LIN {X 0,Y 319.551,Z 618.351,A -85,B 0,C 180,E1 -16134.442,E2 -16134.442} C_VEL
LIN {X 0,Y 320.953,Z 553.396,A -85,B 0,C 180,E1 -16135.793,E2 -16135.793} C_VEL
LIN {X 0,Y 315.824,Z 527.025,A -85,B 0,C 180,E1 -16136.903,E2 -16136.903} C_VEL
LIN {X 0,Y 313.35,Z 517.185,A -85,B 0,C 180,E1 -16137.39,E2 -16137.39} C_VEL
LIN {X 0,Y 311.493,Z 507.907,A -85,B 0,C 180,E1 -16140.123,E2 -16140.123} C_VEL
LIN {X 0,Y 309.031,Z 497.224,A -85,B 0,C 180,E1 -16143.471,E2 -16143.471} C_VEL
LIN {X 0,Y 306.128,Z 486.248,A -85,B 0,C 180,E1 -16147.182,E2 -16147.182} C_VEL
LIN {X 0,Y 305.497,Z 484.053,A -85,B 0,C 180,E1 -16147.997,E2 -16147.997} C_VEL
LIN {X 0,Y 304.829,Z 484.139,A -85,B 0,C 180,E1 -16149.096,E2 -16149.096} C_VEL
LIN {X 0,Y 301.96,Z 484.493,A -85,B 0,C 180,E1 -16150.885,E2 -16150.885} C_VEL
LIN {X 0,Y 299.514,Z 484.803,A -85,B 0,C 180,E1 -16152.335,E2 -16152.335} C_VEL
LIN {X 0,Y 298.446,Z 484.931,A -85,B 0,C 180,E1 -16153.459,E2 -16153.459} C_VEL
LIN {X 0,Y 298.35,Z 484.939,A -85,B 0,C 180,E1 -16153.841,E2 -16153.841} C_VEL
LIN {X 0,Y 298.409,Z 484.934,A -85,B 0,C 180,E1 -16156.921,E2 -16156.921} C_VEL
LIN {X 0,Y 298.405,Z 484.931,A -85,B 0,C 180,E1 -16161.008,E2 -16161.008} C_VEL
LIN {X 0,Y 298.425,Z 484.937,A -85,B 0,C 180,E1 -16163.931,E2 -16163.931} C_VEL
LIN {X 0,Y 298.49,Z 485.123,A -85,B 0,C 180,E1 -16166.405,E2 -16166.405} C_VEL
LIN {X 0,Y 302.37,Z 501.908,A -85,B 0,C 180,E1 -16170.085,E2 -16170.085} C_VEL
LIN {X 0,Y 304.66,Z 513.404,A -85,B 0,C 180,E1 -16172.524,E2 -16172.524} C_VEL
LIN {X 0,Y 303.462,Z 529.943,A -85,B 0,C 180,E1 -16175.727,E2 -16175.727} C_VEL
LIN {X 0,Y 303.246,Z 533.339,A -85,B 0,C 180,E1 -16176.367,E2 -16176.367} C_VEL
LIN {X 0,Y 306.285,Z 559.768,A -85,B 0,C 180,E1 -16177.442,E2 -16177.442} C_VEL
LIN {X 0,Y 303.271,Z 645.533,A -85,B 0,C 180,E1 -16180.365,E2 -16180.365} C_VEL
LIN {X 0,Y 302.635,Z 658.135,A -85,B 0,C 180,E1 -16181.027,E2 -16181.027} C_VEL
LIN {X 0,Y 301.907,Z 671.811,A -85,B 0,C 180,E1 -16182.034,E2 -16182.034} C_VEL
LIN {X 0,Y 300.975,Z 684.908,A -85,B 0,C 180,E1 -16183.311,E2 -16183.311} C_VEL
LIN {X 0,Y 300.064,Z 696.338,A -85,B 0,C 180,E1 -16184.722,E2 -16184.722} C_VEL
LIN {X 0,Y 299.145,Z 707.277,A -85,B 0,C 180,E1 -16186.412,E2 -16186.412} C_VEL
LIN {X 0,Y 298.382,Z 716.255,A -85,B 0,C 180,E1 -16188.106,E2 -16188.106} C_VEL
LIN {X 0,Y 297.71,Z 725.006,A -85,B 0,C 180,E1 -16190.145,E2 -16190.145} C_VEL
LIN {X 0,Y 297.211,Z 732.04,A -85,B 0,C 180,E1 -16192.185,E2 -16192.185} C_VEL
LIN {X 0,Y 296.865,Z 737.87,A -85,B 0,C 180,E1 -16194.322,E2 -16194.322} C_VEL
LIN {X 0,Y 296.754,Z 742.533,A -85,B 0,C 180,E1 -16196.605,E2 -16196.605} C_VEL
LIN {X 0,Y 296.627,Z 745.53,A -85,B 0,C 180,E1 -16198.642,E2 -16198.642} C_VEL
LIN {X 0,Y 296.633,Z 746.97,A -85,B 0,C 180,E1 -16200,E2 -16200} C_VEL
LIN {X 0,Y 296.755,Z 747.956,A -85,B 0,C 180,E1 -16201.357,E2 -16201.357} C_VEL
LIN {X 0,Y 296.931,Z 748.483,A -85,B 0,C 180,E1 -16202.713,E2 -16202.713} C_VEL
LIN {X 0,Y 297.089,Z 748.604,A -85,B 0,C 180,E1 -16204.069,E2 -16204.069} C_VEL
LIN {X 0,Y 297.301,Z 748.296,A -85,B 0,C 180,E1 -16205.426,E2 -16205.426} C_VEL
LIN {X 0,Y 297.711,Z 747.521,A -85,B 0,C 180,E1 -16206.778,E2 -16206.778} C_VEL
LIN {X 0,Y 298.406,Z 746.025,A -85,B 0,C 180,E1 -16208.43,E2 -16208.43} C_VEL
LIN {X 0,Y 299.55,Z 742.622,A -85,B 0,C 180,E1 -16210.818,E2 -16210.818} C_VEL
LIN {X 0,Y 300.846,Z 738.565,A -85,B 0,C 180,E1 -16212.822,E2 -16212.822} C_VEL
LIN {X 0,Y 302.734,Z 732.402,A -85,B 0,C 180,E1 -16215.139,E2 -16215.139} C_VEL
LIN {X 0,Y 304.769,Z 725.583,A -85,B 0,C 180,E1 -16217.098,E2 -16217.098} C_VEL
LIN {X 0,Y 306.644,Z 718.669,A -85,B 0,C 180,E1 -16218.715,E2 -16218.715} C_VEL
LIN {X 0,Y 309.275,Z 708.641,A -85,B 0,C 180,E1 -16220.623,E2 -16220.623} C_VEL
LIN {X 0,Y 311.91,Z 697.136,A -85,B 0,C 180,E1 -16222.343,E2 -16222.343} C_VEL
LIN {X 0,Y 314.257,Z 685.303,A -85,B 0,C 180,E1 -16223.738,E2 -16223.738} C_VEL
LIN {X 0,Y 316.279,Z 674.01,A -85,B 0,C 180,E1 -16224.798,E2 -16224.798} C_VEL
LIN {X 0,Y 318.093,Z 661.718,A -85,B 0,C 180,E1 -16225.696,E2 -16225.696} C_VEL
LIN {X 0,Y 319.7,Z 647.864,A -85,B 0,C 180,E1 -16226.433,E2 -16226.433} C_VEL
LIN {X 0,Y 327.907,Z 571.032,A -85,B 0,C 180,E1 -16229.456,E2 -16229.456} C_VEL
LIN {X 0,Y 327.938,Z 568.4,A -85,B 0,C 180,E1 -16229.628,E2 -16229.628} C_VEL
LIN {X 0,Y 326.362,Z 556.568,A -85,B 0,C 180,E1 -16230.828,E2 -16230.828} C_VEL
LIN {X 0,Y 324.446,Z 544.971,A -85,B 0,C 180,E1 -16232.247,E2 -16232.247} C_VEL
LIN {X 0,Y 322.625,Z 540.593,A -85,B 0,C 180,E1 -16233.189,E2 -16233.189} C_VEL
LIN {X 0,Y 322.019,Z 534.22,A -85,B 0,C 180,E1 -16235.642,E2 -16235.642} C_VEL
LIN {X 0,Y 321.293,Z 529.338,A -85,B 0,C 180,E1 -16238.049,E2 -16238.049} C_VEL
LIN {X 0,Y 320.801,Z 526.352,A -85,B 0,C 180,E1 -16239.934,E2 -16239.934} C_VEL
LIN {X 0,Y 320.418,Z 524.32,A -85,B 0,C 180,E1 -16241.774,E2 -16241.774} C_VEL
LIN {X 0,Y 320.289,Z 522.915,A -85,B 0,C 180,E1 -16243.604,E2 -16243.604} C_VEL
LIN {X 0,Y 320.596,Z 522.275,A -85,B 0,C 180,E1 -16246.337,E2 -16246.337} C_VEL
LIN {X 0,Y 321.718,Z 523.09,A -85,B 0,C 180,E1 -16249.052,E2 -16249.052} C_VEL
LIN {X 0,Y 323.484,Z 525.204,A -85,B 0,C 180,E1 -16251.456,E2 -16251.456} C_VEL
LIN {X 0,Y 324.046,Z 526.038,A -85,B 0,C 180,E1 -16252.067,E2 -16252.067} C_VEL
LIN {X 0,Y 324.345,Z 528.935,A -85,B 0,C 180,E1 -16253.107,E2 -16253.107} C_VEL
LIN {X 0,Y 325.342,Z 539.139,A -85,B 0,C 180,E1 -16255.829,E2 -16255.829} C_VEL
LIN {X 0,Y 325.845,Z 542.951,A -85,B 0,C 180,E1 -16256.666,E2 -16256.666} C_VEL
LIN {X 0,Y 325.078,Z 550.225,A -85,B 0,C 180,E1 -16257.605,E2 -16257.605} C_VEL
LIN {X 0,Y 325.069,Z 563.307,A -85,B 0,C 180,E1 -16258.604,E2 -16258.604} C_VEL
LIN {X 0,Y 314.684,Z 654.608,A -85,B 0,C 180,E1 -16262.345,E2 -16262.345} C_VEL
LIN {X 0,Y 312.854,Z 674.382,A -85,B 0,C 180,E1 -16263.256,E2 -16263.256} C_VEL
LIN {X 0,Y 311.102,Z 688.949,A -85,B 0,C 180,E1 -16264.221,E2 -16264.221} C_VEL
LIN {X 0,Y 309.164,Z 702.373,A -85,B 0,C 180,E1 -16265.407,E2 -16265.407} C_VEL
LIN {X 0,Y 307.546,Z 712.736,A -85,B 0,C 180,E1 -16266.562,E2 -16266.562} C_VEL
LIN {X 0,Y 305.364,Z 724.902,A -85,B 0,C 180,E1 -16268.214,E2 -16268.214} C_VEL
LIN {X 0,Y 303.591,Z 733.816,A -85,B 0,C 180,E1 -16269.68,E2 -16269.68} C_VEL
LIN {X 0,Y 301.64,Z 743.646,A -85,B 0,C 180,E1 -16271.665,E2 -16271.665} C_VEL
LIN {X 0,Y 300.077,Z 751.779,A -85,B 0,C 180,E1 -16273.676,E2 -16273.676} C_VEL
LIN {X 0,Y 298.889,Z 758.364,A -85,B 0,C 180,E1 -16275.705,E2 -16275.705} C_VEL
LIN {X 0,Y 297.841,Z 763.736,A -85,B 0,C 180,E1 -16277.737,E2 -16277.737} C_VEL
LIN {X 0,Y 297.203,Z 767.938,A -85,B 0,C 180,E1 -16279.783,E2 -16279.783} C_VEL
LIN {X 0,Y 296.807,Z 771.086,A -85,B 0,C 180,E1 -16281.831,E2 -16281.831} C_VEL
LIN {X 0,Y 296.594,Z 773.62,A -85,B 0,C 180,E1 -16284.396,E2 -16284.396} C_VEL
LIN {X 0,Y 296.64,Z 774.399,A -85,B 0,C 180,E1 -16285.922,E2 -16285.922} C_VEL
LIN {X 0,Y 296.811,Z 774.874,A -85,B 0,C 180,E1 -16289.998,E2 -16289.998} C_VEL
LIN {X 0,Y 296.673,Z 774.112,A -85,B 0,C 180,E1 -16292.714,E2 -16292.714} C_VEL
LIN {X 0,Y 296.687,Z 771.88,A -85,B 0,C 180,E1 -16295.435,E2 -16295.435} C_VEL
LIN {X 0,Y 296.71,Z 769.242,A -85,B 0,C 180,E1 -16297.484,E2 -16297.484} C_VEL
LIN {X 0,Y 297.057,Z 764.251,A -85,B 0,C 180,E1 -16300.219,E2 -16300.219} C_VEL
LIN {X 0,Y 297.678,Z 759.411,A -85,B 0,C 180,E1 -16302.266,E2 -16302.266} C_VEL
LIN {X 0,Y 298.579,Z 752.32,A -85,B 0,C 180,E1 -16304.655,E2 -16304.655} C_VEL
LIN {X 0,Y 299.825,Z 744.889,A -85,B 0,C 180,E1 -16306.685,E2 -16306.685} C_VEL
LIN {X 0,Y 301.331,Z 735.904,A -85,B 0,C 180,E1 -16308.703,E2 -16308.703} C_VEL
LIN {X 0,Y 302.842,Z 726.968,A -85,B 0,C 180,E1 -16310.369,E2 -16310.369} C_VEL
LIN {X 0,Y 304.77,Z 716.28,A -85,B 0,C 180,E1 -16312.005,E2 -16312.005} C_VEL
LIN {X 0,Y 306.67,Z 703.494,A -85,B 0,C 180,E1 -16313.597,E2 -16313.597} C_VEL
LIN {X 0,Y 308.373,Z 691.684,A -85,B 0,C 180,E1 -16314.755,E2 -16314.755} C_VEL
LIN {X 0,Y 310.052,Z 678.252,A -85,B 0,C 180,E1 -16315.778,E2 -16315.778} C_VEL
LIN {X 0,Y 311.401,Z 664.119,A -85,B 0,C 180,E1 -16316.559,E2 -16316.559} C_VEL
LIN {X 0,Y 312.339,Z 650.423,A -85,B 0,C 180,E1 -16317.059,E2 -16317.059} C_VEL
LIN {X 0,Y 315.103,Z 559.841,A -85,B 0,C 180,E1 -16319.246,E2 -16319.246} C_VEL
LIN {X 0,Y 310.597,Z 527.887,A -85,B 0,C 180,E1 -16320.542,E2 -16320.542} C_VEL
LIN {X 0,Y 308.137,Z 521.44,A -85,B 0,C 180,E1 -16320.991,E2 -16320.991} C_VEL
LIN {X 0,Y 305.142,Z 508.508,A -85,B 0,C 180,E1 -16324.478,E2 -16324.478} C_VEL
LIN {X 0,Y 302.125,Z 497.283,A -85,B 0,C 180,E1 -16327.73,E2 -16327.73} C_VEL
LIN {X 0,Y 299.234,Z 487.6,A -85,B 0,C 180,E1 -16330.761,E2 -16330.761} C_VEL
LIN {X 0,Y 298.441,Z 484.935,A -85,B 0,C 180,E1 -16331.699,E2 -16331.699} C_VEL
LIN {X 0,Y 298.482,Z 484.929,A -85,B 0,C 180,E1 -16335.059,E2 -16335.059} C_VEL
LIN {X 0,Y 298.448,Z 484.932,A -85,B 0,C 180,E1 -16338.896,E2 -16338.896} C_VEL
LIN {X 0,Y 298.462,Z 484.907,A -85,B 0,C 180,E1 -16343.185,E2 -16343.185} C_VEL
LIN {X 0,Y 298.388,Z 484.938,A -85,B 0,C 180,E1 -16347.199,E2 -16347.199} C_VEL
LIN {X 0,Y 298.423,Z 484.938,A -85,B 0,C 180,E1 -16350.613,E2 -16350.613} C_VEL
LIN {X 0,Y 298.482,Z 484.929,A -85,B 0,C 180,E1 -16353.47,E2 -16353.47} C_VEL
LIN {X 0,Y 298.42,Z 484.907,A -85,B 0,C 180,E1 -16356.699,E2 -16356.699} C_VEL
LIN {X 0,Y 298.514,Z 484.918,A -85,B 0,C 180,E1 -16360.755,E2 -16360.755} C_VEL
LIN {X 0,Y 298.582,Z 484.911,A -85,B 0,C 180,E1 -16364.994,E2 -16364.994} C_VEL
LIN {X 0,Y 298.585,Z 484.908,A -85,B 0,C 180,E1 -16369.146,E2 -16369.146} C_VEL
LIN {X 0,Y 298.748,Z 484.896,A -85,B 0,C 180,E1 -16371.886,E2 -16371.886} C_VEL
LIN {X 0,Y 298.652,Z 484.9,A -85,B 0,C 180,E1 -16374.599,E2 -16374.599} C_VEL
LIN {X 0,Y 298.915,Z 484.865,A -85,B 0,C 180,E1 -16378.653,E2 -16378.653} C_VEL
LIN {X 0,Y 298.915,Z 484.875,A -85,B 0,C 180,E1 -16381.347,E2 -16381.347} C_VEL
LIN {X 0,Y 298.787,Z 484.889,A -85,B 0,C 180,E1 -16386.754,E2 -16386.754} C_VEL
LIN {X 0,Y 298.67,Z 484.901,A -85,B 0,C 180,E1 -16389.481,E2 -16389.481} C_VEL
LIN {X 0,Y 298.543,Z 484.911,A -85,B 0,C 180,E1 -16393.616,E2 -16393.616} C_VEL
LIN {X 0,Y 298.539,Z 484.921,A -85,B 0,C 180,E1 -16396.409,E2 -16396.409} C_VEL
LIN {X 0,Y 298.502,Z 484.926,A -85,B 0,C 180,E1 -16399.656,E2 -16399.656} C_VEL
LIN {X 0,Y 298.448,Z 484.932,A -85,B 0,C 180,E1 -16403.599,E2 -16403.599} C_VEL
LIN {X 0,Y 298.481,Z 484.922,A -85,B 0,C 180,E1 -16406.576,E2 -16406.576} C_VEL
LIN {X 0,Y 298.417,Z 484.932,A -85,B 0,C 180,E1 -16409.642,E2 -16409.642} C_VEL
LIN {X 0,Y 298.39,Z 484.938,A -85,B 0,C 180,E1 -16412.801,E2 -16412.801} C_VEL
LIN {X 0,Y 298.459,Z 484.927,A -85,B 0,C 180,E1 -16416.814,E2 -16416.814} C_VEL
LIN {X 0,Y 298.412,Z 484.939,A -85,B 0,C 180,E1 -16421.096,E2 -16421.096} C_VEL
LIN {X 0,Y 298.452,Z 484.93,A -85,B 0,C 180,E1 -16423.117,E2 -16423.117} C_VEL
LIN {X 0,Y 298.461,Z 484.935,A -85,B 0,C 180,E1 -16426.934,E2 -16426.934} C_VEL
LIN {X 0,Y 298.442,Z 484.937,A -85,B 0,C 180,E1 -16431.115,E2 -16431.115} C_VEL
LIN {X 0,Y 298.484,Z 485.1,A -85,B 0,C 180,E1 -16431.397,E2 -16431.397} C_VEL
LIN {X 0,Y 301.365,Z 495.67,A -85,B 0,C 180,E1 -16435.144,E2 -16435.144} C_VEL
LIN {X 0,Y 303.83,Z 505.703,A -85,B 0,C 180,E1 -16438.455,E2 -16438.455} C_VEL
LIN {X 0,Y 306.135,Z 516.337,A -85,B 0,C 180,E1 -16441.737,E2 -16441.737} C_VEL
LIN {X 0,Y 306.408,Z 517.474,A -85,B 0,C 180,E1 -16442.014,E2 -16442.014} C_VEL
LIN {X 0,Y 308.625,Z 523.765,A -85,B 0,C 180,E1 -16442.404,E2 -16442.404} C_VEL
LIN {X 0,Y 314.368,Z 553.15,A -85,B 0,C 180,E1 -16443.695,E2 -16443.695} C_VEL
LIN {X 0,Y 314.608,Z 558.22,A -85,B 0,C 180,E1 -16443.837,E2 -16443.837} C_VEL
LIN {X 0,Y 312.714,Z 632.891,A -85,B 0,C 180,E1 -16445.434,E2 -16445.434} C_VEL
LIN {X 0,Y 312.05,Z 645.796,A -85,B 0,C 180,E1 -16445.954,E2 -16445.954} C_VEL
LIN {X 0,Y 310.947,Z 658.382,A -85,B 0,C 180,E1 -16446.703,E2 -16446.703} C_VEL
LIN {X 0,Y 309.67,Z 670.116,A -85,B 0,C 180,E1 -16447.659,E2 -16447.659} C_VEL
LIN {X 0,Y 308.094,Z 680.821,A -85,B 0,C 180,E1 -16448.771,E2 -16448.771} C_VEL
LIN {X 0,Y 306.4,Z 691.523,A -85,B 0,C 180,E1 -16450.179,E2 -16450.179} C_VEL
LIN {X 0,Y 304.626,Z 701.627,A -85,B 0,C 180,E1 -16451.855,E2 -16451.855} C_VEL
LIN {X 0,Y 302.685,Z 711.162,A -85,B 0,C 180,E1 -16453.824,E2 -16453.824} C_VEL
LIN {X 0,Y 301.155,Z 718.856,A -85,B 0,C 180,E1 -16455.818,E2 -16455.818} C_VEL
LIN {X 0,Y 299.851,Z 725.068,A -85,B 0,C 180,E1 -16457.824,E2 -16457.824} C_VEL
LIN {X 0,Y 298.727,Z 730.051,A -85,B 0,C 180,E1 -16459.839,E2 -16459.839} C_VEL
LIN {X 0,Y 297.849,Z 734.689,A -85,B 0,C 180,E1 -16462.32,E2 -16462.32} C_VEL
LIN {X 0,Y 297.318,Z 737.678,A -85,B 0,C 180,E1 -16464.576,E2 -16464.576} C_VEL
LIN {X 0,Y 296.979,Z 739.854,A -85,B 0,C 180,E1 -16467.289,E2 -16467.289} C_VEL
LIN {X 0,Y 296.86,Z 740.616,A -85,B 0,C 180,E1 -16470.002,E2 -16470.002} C_VEL
LIN {X 0,Y 296.974,Z 739.913,A -85,B 0,C 180,E1 -16472.715,E2 -16472.715} C_VEL
LIN {X 0,Y 297.3,Z 737.786,A -85,B 0,C 180,E1 -16475.428,E2 -16475.428} C_VEL
LIN {X 0,Y 297.909,Z 734.723,A -85,B 0,C 180,E1 -16477.764,E2 -16477.764} C_VEL
LIN {X 0,Y 298.724,Z 730.289,A -85,B 0,C 180,E1 -16480.165,E2 -16480.165} C_VEL
LIN {X 0,Y 299.797,Z 725.361,A -85,B 0,C 180,E1 -16482.182,E2 -16482.182} C_VEL
LIN {X 0,Y 301.071,Z 719.226,A -85,B 0,C 180,E1 -16484.19,E2 -16484.19} C_VEL
LIN {X 0,Y 302.361,Z 712.997,A -85,B 0,C 180,E1 -16485.851,E2 -16485.851} C_VEL
LIN {X 0,Y 303.935,Z 705.561,A -85,B 0,C 180,E1 -16487.496,E2 -16487.496} C_VEL
LIN {X 0,Y 305.642,Z 696.578,A -85,B 0,C 180,E1 -16489.135,E2 -16489.135} C_VEL
LIN {X 0,Y 307.335,Z 685.548,A -85,B 0,C 180,E1 -16490.761,E2 -16490.761} C_VEL
LIN {X 0,Y 309.119,Z 674.402,A -85,B 0,C 180,E1 -16492.034,E2 -16492.034} C_VEL
LIN {X 0,Y 310.429,Z 663.913,A -85,B 0,C 180,E1 -16492.989,E2 -16492.989} C_VEL
LIN {X 0,Y 311.679,Z 651.324,A -85,B 0,C 180,E1 -16493.859,E2 -16493.859} C_VEL
LIN {X 0,Y 312.554,Z 638.179,A -85,B 0,C 180,E1 -16494.495,E2 -16494.495} C_VEL
LIN {X 0,Y 313.085,Z 623.763,A -85,B 0,C 180,E1 -16494.893,E2 -16494.893} C_VEL
LIN {X 0,Y 314.574,Z 554.024,A -85,B 0,C 180,E1 -16496.38,E2 -16496.38} C_VEL
LIN {X 0,Y 309.735,Z 528.951,A -85,B 0,C 180,E1 -16497.468,E2 -16497.468} C_VEL
LIN {X 0,Y 307.563,Z 520.38,A -85,B 0,C 180,E1 -16497.908,E2 -16497.908} C_VEL
LIN {X 0,Y 306.255,Z 517.123,A -85,B 0,C 180,E1 -16498.156,E2 -16498.156} C_VEL
LIN {X 0,Y 303.917,Z 506.074,A -85,B 0,C 180,E1 -16501.55,E2 -16501.55} C_VEL
LIN {X 0,Y 301.627,Z 496.65,A -85,B 0,C 180,E1 -16504.647,E2 -16504.647} C_VEL
LIN {X 0,Y 299.021,Z 486.978,A -85,B 0,C 180,E1 -16508.05,E2 -16508.05} C_VEL
LIN {X 0,Y 298.421,Z 484.934,A -85,B 0,C 180,E1 -16508.881,E2 -16508.881} C_VEL
LIN {X 0,Y 298.405,Z 484.94,A -85,B 0,C 180,E1 -16513.104,E2 -16513.104} C_VEL
LIN {X 0,Y 298.35,Z 484.939,A -85,B 0,C 180,E1 -16513.841,E2 -16513.841} C_VEL
LIN {X 0,Y 297.656,Z 485.028,A -85,B 0,C 180,E1 -16514.968,E2 -16514.968} C_VEL
LIN {X 0,Y 294.801,Z 485.384,A -85,B 0,C 180,E1 -16516.804,E2 -16516.804} C_VEL
LIN {X 0,Y 292.413,Z 485.683,A -85,B 0,C 180,E1 -16518.294,E2 -16518.294} C_VEL
LIN {X 0,Y 291.413,Z 485.809,A -85,B 0,C 180,E1 -16519.448,E2 -16519.448} C_VEL
LIN {X 0,Y 291.343,Z 485.815,A -85,B 0,C 180,E1 -16519.838,E2 -16519.838} C_VEL
LIN {X 0,Y 291.411,Z 485.801,A -85,B 0,C 180,E1 -16522.92,E2 -16522.92} C_VEL
LIN {X 0,Y 291.43,Z 485.926,A -85,B 0,C 180,E1 -16526.036,E2 -16526.036} C_VEL
LIN {X 0,Y 295.585,Z 503.96,A -85,B 0,C 180,E1 -16530.045,E2 -16530.045} C_VEL
LIN {X 0,Y 297.659,Z 513.957,A -85,B 0,C 180,E1 -16532.204,E2 -16532.204} C_VEL
LIN {X 0,Y 297.115,Z 523.099,A -85,B 0,C 180,E1 -16534.011,E2 -16534.011} C_VEL
LIN {X 0,Y 296.323,Z 533.48,A -85,B 0,C 180,E1 -16536.036,E2 -16536.036} C_VEL
LIN {X 0,Y 299.087,Z 557.753,A -85,B 0,C 180,E1 -16537.06,E2 -16537.06} C_VEL
LIN {X 0,Y 299.299,Z 562.384,A -85,B 0,C 180,E1 -16537.24,E2 -16537.24} C_VEL
LIN {X 0,Y 296.234,Z 645.935,A -85,B 0,C 180,E1 -16540.195,E2 -16540.195} C_VEL
LIN {X 0,Y 295.572,Z 659.126,A -85,B 0,C 180,E1 -16540.916,E2 -16540.916} C_VEL
LIN {X 0,Y 294.821,Z 672.643,A -85,B 0,C 180,E1 -16541.947,E2 -16541.947} C_VEL
LIN {X 0,Y 293.966,Z 684.253,A -85,B 0,C 180,E1 -16543.099,E2 -16543.099} C_VEL
LIN {X 0,Y 293.055,Z 695.729,A -85,B 0,C 180,E1 -16544.526,E2 -16544.526} C_VEL
LIN {X 0,Y 292.197,Z 705.892,A -85,B 0,C 180,E1 -16546.082,E2 -16546.082} C_VEL
LIN {X 0,Y 291.382,Z 715.151,A -85,B 0,C 180,E1 -16547.816,E2 -16547.816} C_VEL
LIN {X 0,Y 290.692,Z 724.226,A -85,B 0,C 180,E1 -16549.905,E2 -16549.905} C_VEL
LIN {X 0,Y 290.142,Z 731.435,A -85,B 0,C 180,E1 -16551.994,E2 -16551.994} C_VEL
LIN {X 0,Y 289.779,Z 738.074,A -85,B 0,C 180,E1 -16554.433,E2 -16554.433} C_VEL
LIN {X 0,Y 289.667,Z 742.371,A -85,B 0,C 180,E1 -16556.522,E2 -16556.522} C_VEL
LIN {X 0,Y 289.544,Z 745.542,A -85,B 0,C 180,E1 -16558.609,E2 -16558.609} C_VEL
LIN {X 0,Y 289.546,Z 747.065,A -85,B 0,C 180,E1 -16560,E2 -16560} C_VEL
LIN {X 0,Y 289.669,Z 748.171,A -85,B 0,C 180,E1 -16561.39,E2 -16561.39} C_VEL
LIN {X 0,Y 289.849,Z 748.817,A -85,B 0,C 180,E1 -16562.779,E2 -16562.779} C_VEL
LIN {X 0,Y 290.023,Z 749.021,A -85,B 0,C 180,E1 -16564.169,E2 -16564.169} C_VEL
LIN {X 0,Y 290.266,Z 748.82,A -85,B 0,C 180,E1 -16565.558,E2 -16565.558} C_VEL
LIN {X 0,Y 290.707,Z 748.19,A -85,B 0,C 180,E1 -16566.943,E2 -16566.943} C_VEL
LIN {X 0,Y 291.403,Z 746.85,A -85,B 0,C 180,E1 -16568.563,E2 -16568.563} C_VEL
LIN {X 0,Y 292.652,Z 743.632,A -85,B 0,C 180,E1 -16571.076,E2 -16571.076} C_VEL
LIN {X 0,Y 294.049,Z 739.813,A -85,B 0,C 180,E1 -16573.124,E2 -16573.124} C_VEL
LIN {X 0,Y 295.717,Z 734.817,A -85,B 0,C 180,E1 -16575.155,E2 -16575.155} C_VEL
LIN {X 0,Y 298.189,Z 727.329,A -85,B 0,C 180,E1 -16577.488,E2 -16577.488} C_VEL
LIN {X 0,Y 300.171,Z 720.766,A -85,B 0,C 180,E1 -16579.134,E2 -16579.134} C_VEL
LIN {X 0,Y 302.447,Z 712.881,A -85,B 0,C 180,E1 -16580.754,E2 -16580.754} C_VEL
LIN {X 0,Y 305.407,Z 701.466,A -85,B 0,C 180,E1 -16582.635,E2 -16582.635} C_VEL
LIN {X 0,Y 307.883,Z 690.626,A -85,B 0,C 180,E1 -16584.063,E2 -16584.063} C_VEL
LIN {X 0,Y 310.271,Z 678.661,A -85,B 0,C 180,E1 -16585.311,E2 -16585.311} C_VEL
LIN {X 0,Y 312.693,Z 664.342,A -85,B 0,C 180,E1 -16586.442,E2 -16586.442} C_VEL
LIN {X 0,Y 314.368,Z 651.683,A -85,B 0,C 180,E1 -16587.187,E2 -16587.187} C_VEL
LIN {X 0,Y 321.466,Z 589.165,A -85,B 0,C 180,E1 -16589.738,E2 -16589.738} C_VEL
LIN {X 0,Y 323.605,Z 571.225,A -85,B 0,C 180,E1 -16590.478,E2 -16590.478} C_VEL
LIN {X 0,Y 322.194,Z 558.888,A -85,B 0,C 180,E1 -16591.79,E2 -16591.79} C_VEL
LIN {X 0,Y 320.829,Z 549.545,A -85,B 0,C 180,E1 -16592.987,E2 -16592.987} C_VEL
LIN {X 0,Y 318.353,Z 543.626,A -85,B 0,C 180,E1 -16594.409,E2 -16594.409} C_VEL
LIN {X 0,Y 317.415,Z 541.077,A -85,B 0,C 180,E1 -16595.147,E2 -16595.147} C_VEL
LIN {X 0,Y 316.927,Z 535.764,A -85,B 0,C 180,E1 -16597.674,E2 -16597.674} C_VEL
LIN {X 0,Y 316.5,Z 531.955,A -85,B 0,C 180,E1 -16600.087,E2 -16600.087} C_VEL
LIN {X 0,Y 316.268,Z 529.283,A -85,B 0,C 180,E1 -16602.833,E2 -16602.833} C_VEL
LIN {X 0,Y 316.457,Z 528.292,A -85,B 0,C 180,E1 -16605.289,E2 -16605.289} C_VEL
LIN {X 0,Y 316.953,Z 528.33,A -85,B 0,C 180,E1 -16607.031,E2 -16607.031} C_VEL
LIN {X 0,Y 317.802,Z 528.966,A -85,B 0,C 180,E1 -16608.754,E2 -16608.754} C_VEL
LIN {X 0,Y 318.974,Z 530.255,A -85,B 0,C 180,E1 -16610.458,E2 -16610.458} C_VEL
LIN {X 0,Y 319.801,Z 531.312,A -85,B 0,C 180,E1 -16611.437,E2 -16611.437} C_VEL
LIN {X 0,Y 320.303,Z 532.714,A -85,B 0,C 180,E1 -16612.176,E2 -16612.176} C_VEL
LIN {X 0,Y 320.817,Z 541.692,A -85,B 0,C 180,E1 -16614.732,E2 -16614.732} C_VEL
LIN {X 0,Y 321.405,Z 546.766,A -85,B 0,C 180,E1 -16615.943,E2 -16615.943} C_VEL
LIN {X 0,Y 321.098,Z 550.829,A -85,B 0,C 180,E1 -16616.481,E2 -16616.481} C_VEL
LIN {X 0,Y 320.981,Z 564.626,A -85,B 0,C 180,E1 -16617.592,E2 -16617.592} C_VEL
LIN {X 0,Y 309.564,Z 658.052,A -85,B 0,C 180,E1 -16621.524,E2 -16621.524} C_VEL
LIN {X 0,Y 307.91,Z 673.964,A -85,B 0,C 180,E1 -16622.284,E2 -16622.284} C_VEL
LIN {X 0,Y 306.034,Z 687.748,A -85,B 0,C 180,E1 -16623.211,E2 -16623.211} C_VEL
LIN {X 0,Y 304.003,Z 700.697,A -85,B 0,C 180,E1 -16624.347,E2 -16624.347} C_VEL
LIN {X 0,Y 301.959,Z 712.076,A -85,B 0,C 180,E1 -16625.623,E2 -16625.623} C_VEL
LIN {X 0,Y 299.709,Z 723.784,A -85,B 0,C 180,E1 -16627.236,E2 -16627.236} C_VEL
LIN {X 0,Y 297.503,Z 733.608,A -85,B 0,C 180,E1 -16628.882,E2 -16628.882} C_VEL
LIN {X 0,Y 295.331,Z 743.384,A -85,B 0,C 180,E1 -16630.899,E2 -16630.899} C_VEL
LIN {X 0,Y 293.603,Z 751.4,A -85,B 0,C 180,E1 -16632.947,E2 -16632.947} C_VEL
LIN {X 0,Y 292.4,Z 756.984,A -85,B 0,C 180,E1 -16634.668,E2 -16634.668} C_VEL
LIN {X 0,Y 291.288,Z 762.517,A -85,B 0,C 180,E1 -16636.748,E2 -16636.748} C_VEL
LIN {X 0,Y 290.394,Z 766.89,A -85,B 0,C 180,E1 -16638.835,E2 -16638.835} C_VEL
LIN {X 0,Y 290,Z 769.196,A -85,B 0,C 180,E1 -16640.231,E2 -16640.231} C_VEL
LIN {X 0,Y 289.739,Z 771.067,A -85,B 0,C 180,E1 -16641.63,E2 -16641.63} C_VEL
LIN {X 0,Y 289.571,Z 772.52,A -85,B 0,C 180,E1 -16643.028,E2 -16643.028} C_VEL
LIN {X 0,Y 289.517,Z 773.509,A -85,B 0,C 180,E1 -16644.426,E2 -16644.426} C_VEL
LIN {X 0,Y 289.551,Z 774.063,A -85,B 0,C 180,E1 -16645.822,E2 -16645.822} C_VEL
LIN {X 0,Y 289.721,Z 774.465,A -85,B 0,C 180,E1 -16649.998,E2 -16649.998} C_VEL
LIN {X 0,Y 289.595,Z 773.702,A -85,B 0,C 180,E1 -16652.78,E2 -16652.78} C_VEL
LIN {X 0,Y 289.603,Z 771.467,A -85,B 0,C 180,E1 -16655.569,E2 -16655.569} C_VEL
LIN {X 0,Y 289.704,Z 767.71,A -85,B 0,C 180,E1 -16658.368,E2 -16658.368} C_VEL
LIN {X 0,Y 290.166,Z 762.343,A -85,B 0,C 180,E1 -16661.171,E2 -16661.171} C_VEL
LIN {X 0,Y 290.924,Z 757.106,A -85,B 0,C 180,E1 -16663.265,E2 -16663.265} C_VEL
LIN {X 0,Y 291.976,Z 749.695,A -85,B 0,C 180,E1 -16665.673,E2 -16665.673} C_VEL
LIN {X 0,Y 293.417,Z 741.658,A -85,B 0,C 180,E1 -16667.78,E2 -16667.78} C_VEL
LIN {X 0,Y 295.122,Z 732.073,A -85,B 0,C 180,E1 -16669.835,E2 -16669.835} C_VEL
LIN {X 0,Y 297.152,Z 721.401,A -85,B 0,C 180,E1 -16671.686,E2 -16671.686} C_VEL
LIN {X 0,Y 299.123,Z 709.562,A -85,B 0,C 180,E1 -16673.356,E2 -16673.356} C_VEL
LIN {X 0,Y 300.93,Z 698.052,A -85,B 0,C 180,E1 -16674.661,E2 -16674.661} C_VEL
LIN {X 0,Y 302.815,Z 684.3,A -85,B 0,C 180,E1 -16675.886,E2 -16675.886} C_VEL
LIN {X 0,Y 304.381,Z 670.327,A -85,B 0,C 180,E1 -16676.804,E2 -16676.804} C_VEL
LIN {X 0,Y 305.556,Z 656.545,A -85,B 0,C 180,E1 -16677.432,E2 -16677.432} C_VEL
LIN {X 0,Y 306.33,Z 637.875,A -85,B 0,C 180,E1 -16677.96,E2 -16677.96} C_VEL
LIN {X 0,Y 308.802,Z 560.723,A -85,B 0,C 180,E1 -16679.835,E2 -16679.835} C_VEL
LIN {X 0,Y 304.609,Z 530.259,A -85,B 0,C 180,E1 -16681.101,E2 -16681.101} C_VEL
LIN {X 0,Y 300.931,Z 521.374,A -85,B 0,C 180,E1 -16681.764,E2 -16681.764} C_VEL
LIN {X 0,Y 297.998,Z 508.763,A -85,B 0,C 180,E1 -16685.293,E2 -16685.293} C_VEL
LIN {X 0,Y 294.952,Z 497.652,A -85,B 0,C 180,E1 -16688.657,E2 -16688.657} C_VEL
LIN {X 0,Y 292.104,Z 488.128,A -85,B 0,C 180,E1 -16691.767,E2 -16691.767} C_VEL
LIN {X 0,Y 291.41,Z 485.811,A -85,B 0,C 180,E1 -16692.587,E2 -16692.587} C_VEL
LIN {X 0,Y 291.393,Z 485.81,A -85,B 0,C 180,E1 -16696.346,E2 -16696.346} C_VEL
LIN {X 0,Y 291.405,Z 485.803,A -85,B 0,C 180,E1 -16700.509,E2 -16700.509} C_VEL
LIN {X 0,Y 291.425,Z 485.786,A -85,B 0,C 180,E1 -16702.922,E2 -16702.922} C_VEL
LIN {X 0,Y 291.336,Z 485.811,A -85,B 0,C 180,E1 -16706.301,E2 -16706.301} C_VEL
LIN {X 0,Y 291.378,Z 485.813,A -85,B 0,C 180,E1 -16710.259,E2 -16710.259} C_VEL
LIN {X 0,Y 291.41,Z 485.812,A -85,B 0,C 180,E1 -16714.272,E2 -16714.272} C_VEL
LIN {X 0,Y 291.364,Z 485.779,A -85,B 0,C 180,E1 -16717.298,E2 -16717.298} C_VEL
LIN {X 0,Y 291.447,Z 485.793,A -85,B 0,C 180,E1 -16720.27,E2 -16720.27} C_VEL
LIN {X 0,Y 291.544,Z 485.785,A -85,B 0,C 180,E1 -16724.623,E2 -16724.623} C_VEL
LIN {X 0,Y 291.528,Z 485.786,A -85,B 0,C 180,E1 -16728.88,E2 -16728.88} C_VEL
LIN {X 0,Y 291.698,Z 485.774,A -85,B 0,C 180,E1 -16731.688,E2 -16731.688} C_VEL
LIN {X 0,Y 291.622,Z 485.774,A -85,B 0,C 180,E1 -16734.468,E2 -16734.468} C_VEL
LIN {X 0,Y 291.881,Z 485.741,A -85,B 0,C 180,E1 -16738.62,E2 -16738.62} C_VEL
LIN {X 0,Y 291.881,Z 485.751,A -85,B 0,C 180,E1 -16741.38,E2 -16741.38} C_VEL
LIN {X 0,Y 291.736,Z 485.766,A -85,B 0,C 180,E1 -16746.918,E2 -16746.918} C_VEL
LIN {X 0,Y 291.619,Z 485.78,A -85,B 0,C 180,E1 -16749.712,E2 -16749.712} C_VEL
LIN {X 0,Y 291.512,Z 485.788,A -85,B 0,C 180,E1 -16753.951,E2 -16753.951} C_VEL
LIN {X 0,Y 291.477,Z 485.796,A -85,B 0,C 180,E1 -16756.819,E2 -16756.819} C_VEL
LIN {X 0,Y 291.441,Z 485.806,A -85,B 0,C 180,E1 -16759.876,E2 -16759.876} C_VEL
LIN {X 0,Y 291.391,Z 485.813,A -85,B 0,C 180,E1 -16764.206,E2 -16764.206} C_VEL
LIN {X 0,Y 291.416,Z 485.806,A -85,B 0,C 180,E1 -16767.272,E2 -16767.272} C_VEL
LIN {X 0,Y 291.333,Z 485.812,A -85,B 0,C 180,E1 -16770.438,E2 -16770.438} C_VEL
LIN {X 0,Y 291.339,Z 485.812,A -85,B 0,C 180,E1 -16773.699,E2 -16773.699} C_VEL
LIN {X 0,Y 291.391,Z 485.807,A -85,B 0,C 180,E1 -16777.262,E2 -16777.262} C_VEL
LIN {X 0,Y 291.37,Z 485.813,A -85,B 0,C 180,E1 -16780.637,E2 -16780.637} C_VEL
LIN {X 0,Y 291.347,Z 485.822,A -85,B 0,C 180,E1 -16784.391,E2 -16784.391} C_VEL
LIN {X 0,Y 291.383,Z 485.812,A -85,B 0,C 180,E1 -16788.392,E2 -16788.392} C_VEL
LIN {X 0,Y 291.428,Z 485.951,A -85,B 0,C 180,E1 -16790.508,E2 -16790.508} C_VEL
LIN {X 0,Y 294.285,Z 496.213,A -85,B 0,C 180,E1 -16794.29,E2 -16794.29} C_VEL
LIN {X 0,Y 296.856,Z 506.567,A -85,B 0,C 180,E1 -16797.814,E2 -16797.814} C_VEL
LIN {X 0,Y 299.213,Z 517.374,A -85,B 0,C 180,E1 -16801.224,E2 -16801.224} C_VEL
LIN {X 0,Y 302.549,Z 525.689,A -85,B 0,C 180,E1 -16801.807,E2 -16801.807} C_VEL
LIN {X 0,Y 307.639,Z 551.695,A -85,B 0,C 180,E1 -16802.994,E2 -16802.994} C_VEL
LIN {X 0,Y 308.385,Z 556.945,A -85,B 0,C 180,E1 -16803.196,E2 -16803.196} C_VEL
LIN {X 0,Y 306.367,Z 632.755,A -85,B 0,C 180,E1 -16804.845,E2 -16804.845} C_VEL
LIN {X 0,Y 305.675,Z 645.81,A -85,B 0,C 180,E1 -16805.374,E2 -16805.374} C_VEL
LIN {X 0,Y 304.485,Z 659.03,A -85,B 0,C 180,E1 -16806.178,E2 -16806.178} C_VEL
LIN {X 0,Y 303.135,Z 670.686,A -85,B 0,C 180,E1 -16807.151,E2 -16807.151} C_VEL
LIN {X 0,Y 301.514,Z 681.34,A -85,B 0,C 180,E1 -16808.285,E2 -16808.285} C_VEL
LIN {X 0,Y 299.841,Z 691.511,A -85,B 0,C 180,E1 -16809.647,E2 -16809.647} C_VEL
LIN {X 0,Y 298.281,Z 700.301,A -85,B 0,C 180,E1 -16811.099,E2 -16811.099} C_VEL
LIN {X 0,Y 296.567,Z 708.683,A -85,B 0,C 180,E1 -16812.771,E2 -16812.771} C_VEL
LIN {X 0,Y 294.809,Z 716.894,A -85,B 0,C 180,E1 -16814.8,E2 -16814.8} C_VEL
LIN {X 0,Y 293.44,Z 723.539,A -85,B 0,C 180,E1 -16816.85,E2 -16816.85} C_VEL
LIN {X 0,Y 292.109,Z 728.913,A -85,B 0,C 180,E1 -16818.905,E2 -16818.905} C_VEL
LIN {X 0,Y 291.184,Z 733.175,A -85,B 0,C 180,E1 -16820.976,E2 -16820.976} C_VEL
LIN {X 0,Y 290.626,Z 736.442,A -85,B 0,C 180,E1 -16823.057,E2 -16823.057} C_VEL
LIN {X 0,Y 290.023,Z 739.358,A -85,B 0,C 180,E1 -16825.833,E2 -16825.833} C_VEL
LIN {X 0,Y 289.791,Z 740.82,A -85,B 0,C 180,E1 -16828.612,E2 -16828.612} C_VEL
LIN {X 0,Y 289.79,Z 740.855,A -85,B 0,C 180,E1 -16831.391,E2 -16831.391} C_VEL
LIN {X 0,Y 290.009,Z 739.44,A -85,B 0,C 180,E1 -16834.171,E2 -16834.171} C_VEL
LIN {X 0,Y 290.597,Z 736.577,A -85,B 0,C 180,E1 -16836.947,E2 -16836.947} C_VEL
LIN {X 0,Y 291.186,Z 733.362,A -85,B 0,C 180,E1 -16839.028,E2 -16839.028} C_VEL
LIN {X 0,Y 292.095,Z 729.158,A -85,B 0,C 180,E1 -16841.1,E2 -16841.1} C_VEL
LIN {X 0,Y 293.517,Z 722.875,A -85,B 0,C 180,E1 -16843.502,E2 -16843.502} C_VEL
LIN {X 0,Y 295.112,Z 716.05,A -85,B 0,C 180,E1 -16845.542,E2 -16845.542} C_VEL
LIN {X 0,Y 296.464,Z 709.156,A -85,B 0,C 180,E1 -16847.239,E2 -16847.239} C_VEL
LIN {X 0,Y 298.211,Z 700.876,A -85,B 0,C 180,E1 -16848.91,E2 -16848.91} C_VEL
LIN {X 0,Y 299.998,Z 690.753,A -85,B 0,C 180,E1 -16850.575,E2 -16850.575} C_VEL
LIN {X 0,Y 301.613,Z 680.806,A -85,B 0,C 180,E1 -16851.891,E2 -16851.891} C_VEL
LIN {X 0,Y 303.274,Z 670.017,A -85,B 0,C 180,E1 -16853.022,E2 -16853.022} C_VEL
LIN {X 0,Y 304.769,Z 657.04,A -85,B 0,C 180,E1 -16854.073,E2 -16854.073} C_VEL
LIN {X 0,Y 305.827,Z 643.78,A -85,B 0,C 180,E1 -16854.843,E2 -16854.843} C_VEL
LIN {X 0,Y 306.566,Z 630.377,A -85,B 0,C 180,E1 -16855.323,E2 -16855.323} C_VEL
LIN {X 0,Y 308.344,Z 555.195,A -85,B 0,C 180,E1 -16856.967,E2 -16856.967} C_VEL
LIN {X 0,Y 303.165,Z 528.478,A -85,B 0,C 180,E1 -16858.172,E2 -16858.172} C_VEL
LIN {X 0,Y 301.723,Z 523.23,A -85,B 0,C 180,E1 -16858.464,E2 -16858.464} C_VEL
LIN {X 0,Y 299.139,Z 517.188,A -85,B 0,C 180,E1 -16858.933,E2 -16858.933} C_VEL
LIN {X 0,Y 296.619,Z 505.596,A -85,B 0,C 180,E1 -16862.627,E2 -16862.627} C_VEL
LIN {X 0,Y 294.162,Z 495.606,A -85,B 0,C 180,E1 -16866.056,E2 -16866.056} C_VEL
LIN {X 0,Y 291.377,Z 485.818,A -85,B 0,C 180,E1 -16869.72,E2 -16869.72} C_VEL
LIN {X 0,Y 291.305,Z 485.817,A -85,B 0,C 180,E1 -16873.83,E2 -16873.83} C_VEL
LIN {X 0,Y 291.326,Z 485.811,A -85,B 0,C 180,E1 -16877.508,E2 -16877.508} C_VEL
LIN {X 0,Y 291.343,Z 485.815,A -85,B 0,C 180,E1 -16879.838,E2 -16879.838} C_VEL
LIN {X 0,Y 290.69,Z 485.898,A -85,B 0,C 180,E1 -16880.607,E2 -16880.607} C_VEL
LIN {X 0,Y 287.872,Z 486.248,A -85,B 0,C 180,E1 -16881.813,E2 -16881.813} C_VEL
LIN {X 0,Y 285.014,Z 486.603,A -85,B 0,C 180,E1 -16883.042,E2 -16883.042} C_VEL
LIN {X 0,Y 284.332,Z 486.688,A -85,B 0,C 180,E1 -16883.837,E2 -16883.837} C_VEL
LIN {X 0,Y 284.345,Z 486.698,A -85,B 0,C 180,E1 -16885.653,E2 -16885.653} C_VEL
LIN {X 0,Y 288.401,Z 504.281,A -85,B 0,C 180,E1 -16889.625,E2 -16889.625} C_VEL
LIN {X 0,Y 290.559,Z 514.435,A -85,B 0,C 180,E1 -16891.857,E2 -16891.857} C_VEL
LIN {X 0,Y 290.648,Z 518.271,A -85,B 0,C 180,E1 -16892.649,E2 -16892.649} C_VEL
LIN {X 0,Y 289.383,Z 533.782,A -85,B 0,C 180,E1 -16895.719,E2 -16895.719} C_VEL
LIN {X 0,Y 292.355,Z 559.642,A -85,B 0,C 180,E1 -16896.847,E2 -16896.847} C_VEL
LIN {X 0,Y 289.193,Z 646.323,A -85,B 0,C 180,E1 -16900.016,E2 -16900.016} C_VEL
LIN {X 0,Y 288.49,Z 660.097,A -85,B 0,C 180,E1 -16900.799,E2 -16900.799} C_VEL
LIN {X 0,Y 287.721,Z 673.842,A -85,B 0,C 180,E1 -16901.891,E2 -16901.891} C_VEL
LIN {X 0,Y 286.666,Z 686.793,A -85,B 0,C 180,E1 -16903.257,E2 -16903.257} C_VEL
LIN {X 0,Y 285.915,Z 696.249,A -85,B 0,C 180,E1 -16904.495,E2 -16904.495} C_VEL
LIN {X 0,Y 285.083,Z 706.35,A -85,B 0,C 180,E1 -16906.092,E2 -16906.092} C_VEL
LIN {X 0,Y 284.153,Z 717.245,A -85,B 0,C 180,E1 -16908.226,E2 -16908.226} C_VEL
LIN {X 0,Y 283.462,Z 725.919,A -85,B 0,C 180,E1 -16910.366,E2 -16910.366} C_VEL
LIN {X 0,Y 282.988,Z 732.926,A -85,B 0,C 180,E1 -16912.508,E2 -16912.508} C_VEL
LIN {X 0,Y 282.705,Z 737.637,A -85,B 0,C 180,E1 -16914.293,E2 -16914.293} C_VEL
LIN {X 0,Y 282.583,Z 742.156,A -85,B 0,C 180,E1 -16916.435,E2 -16916.435} C_VEL
LIN {X 0,Y 282.463,Z 745.51,A -85,B 0,C 180,E1 -16918.574,E2 -16918.574} C_VEL
LIN {X 0,Y 282.462,Z 747.144,A -85,B 0,C 180,E1 -16920,E2 -16920} C_VEL
LIN {X 0,Y 282.585,Z 748.328,A -85,B 0,C 180,E1 -16921.425,E2 -16921.425} C_VEL
LIN {X 0,Y 282.771,Z 749.105,A -85,B 0,C 180,E1 -16922.849,E2 -16922.849} C_VEL
LIN {X 0,Y 282.962,Z 749.441,A -85,B 0,C 180,E1 -16924.273,E2 -16924.273} C_VEL
LIN {X 0,Y 283.235,Z 749.326,A -85,B 0,C 180,E1 -16925.696,E2 -16925.696} C_VEL
LIN {X 0,Y 283.707,Z 748.795,A -85,B 0,C 180,E1 -16927.115,E2 -16927.115} C_VEL
LIN {X 0,Y 284.377,Z 747.726,A -85,B 0,C 180,E1 -16928.672,E2 -16928.672} C_VEL
LIN {X 0,Y 285.759,Z 744.629,A -85,B 0,C 180,E1 -16931.347,E2 -16931.347} C_VEL
LIN {X 0,Y 287.254,Z 740.996,A -85,B 0,C 180,E1 -16933.44,E2 -16933.44} C_VEL
LIN {X 0,Y 289.033,Z 736.271,A -85,B 0,C 180,E1 -16935.514,E2 -16935.514} C_VEL
LIN {X 0,Y 291.251,Z 730.284,A -85,B 0,C 180,E1 -16937.555,E2 -16937.555} C_VEL
LIN {X 0,Y 293.707,Z 722.803,A -85,B 0,C 180,E1 -16939.572,E2 -16939.572} C_VEL
LIN {X 0,Y 296.633,Z 713.656,A -85,B 0,C 180,E1 -16941.545,E2 -16941.545} C_VEL
LIN {X 0,Y 299.55,Z 703.304,A -85,B 0,C 180,E1 -16943.313,E2 -16943.313} C_VEL
LIN {X 0,Y 302.419,Z 691.704,A -85,B 0,C 180,E1 -16944.893,E2 -16944.893} C_VEL
LIN {X 0,Y 304.972,Z 680.086,A -85,B 0,C 180,E1 -16946.15,E2 -16946.15} C_VEL
LIN {X 0,Y 307.348,Z 667.324,A -85,B 0,C 180,E1 -16947.215,E2 -16947.215} C_VEL
LIN {X 0,Y 309.322,Z 654.153,A -85,B 0,C 180,E1 -16948.036,E2 -16948.036} C_VEL
LIN {X 0,Y 312.485,Z 627.682,A -85,B 0,C 180,E1 -16949.194,E2 -16949.194} C_VEL
LIN {X 0,Y 319.378,Z 573.18,A -85,B 0,C 180,E1 -16951.46,E2 -16951.46} C_VEL
LIN {X 0,Y 318.254,Z 561.572,A -85,B 0,C 180,E1 -16952.762,E2 -16952.762} C_VEL
LIN {X 0,Y 317.353,Z 554.239,A -85,B 0,C 180,E1 -16953.738,E2 -16953.738} C_VEL
LIN {X 0,Y 315.101,Z 548.401,A -85,B 0,C 180,E1 -16955.217,E2 -16955.217} C_VEL
LIN {X 0,Y 312.518,Z 542.346,A -85,B 0,C 180,E1 -16957.24,E2 -16957.24} C_VEL
LIN {X 0,Y 312.314,Z 539.252,A -85,B 0,C 180,E1 -16959.056,E2 -16959.056} C_VEL
LIN {X 0,Y 312.217,Z 537.011,A -85,B 0,C 180,E1 -16960.752,E2 -16960.752} C_VEL
LIN {X 0,Y 312.2,Z 535.442,A -85,B 0,C 180,E1 -16962.48,E2 -16962.48} C_VEL
LIN {X 0,Y 312.362,Z 534.451,A -85,B 0,C 180,E1 -16964.226,E2 -16964.226} C_VEL
LIN {X 0,Y 312.759,Z 534.207,A -85,B 0,C 180,E1 -16965.978,E2 -16965.978} C_VEL
LIN {X 0,Y 313.467,Z 534.536,A -85,B 0,C 180,E1 -16967.73,E2 -16967.73} C_VEL
LIN {X 0,Y 314.645,Z 535.658,A -85,B 0,C 180,E1 -16969.626,E2 -16969.626} C_VEL
LIN {X 0,Y 316.168,Z 537.674,A -85,B 0,C 180,E1 -16971.506,E2 -16971.506} C_VEL
LIN {X 0,Y 316.322,Z 540.147,A -85,B 0,C 180,E1 -16972.38,E2 -16972.38} C_VEL
LIN {X 0,Y 316.9,Z 549.173,A -85,B 0,C 180,E1 -16974.845,E2 -16974.845} C_VEL
LIN {X 0,Y 317.407,Z 551.558,A -85,B 0,C 180,E1 -16975.269,E2 -16975.269} C_VEL
LIN {X 0,Y 317.437,Z 557.447,A -85,B 0,C 180,E1 -16975.851,E2 -16975.851} C_VEL
LIN {X 0,Y 317.066,Z 567.077,A -85,B 0,C 180,E1 -16976.597,E2 -16976.597} C_VEL
LIN {X 0,Y 304.616,Z 661.333,A -85,B 0,C 180,E1 -16980.64,E2 -16980.64} C_VEL
LIN {X 0,Y 302.874,Z 675.885,A -85,B 0,C 180,E1 -16981.405,E2 -16981.405} C_VEL
LIN {X 0,Y 300.523,Z 690.906,A -85,B 0,C 180,E1 -16982.491,E2 -16982.491} C_VEL
LIN {X 0,Y 298.216,Z 703.297,A -85,B 0,C 180,E1 -16983.675,E2 -16983.675} C_VEL
LIN {X 0,Y 296.013,Z 714.293,A -85,B 0,C 180,E1 -16984.993,E2 -16984.993} C_VEL
LIN {X 0,Y 293.422,Z 725.948,A -85,B 0,C 180,E1 -16986.719,E2 -16986.719} C_VEL
LIN {X 0,Y 291.071,Z 735.322,A -85,B 0,C 180,E1 -16988.393,E2 -16988.393} C_VEL
LIN {X 0,Y 288.74,Z 744.635,A -85,B 0,C 180,E1 -16990.445,E2 -16990.445} C_VEL
LIN {X 0,Y 286.576,Z 753.464,A -85,B 0,C 180,E1 -16992.883,E2 -16992.883} C_VEL
LIN {X 0,Y 285.173,Z 759.547,A -85,B 0,C 180,E1 -16995.001,E2 -16995.001} C_VEL
LIN {X 0,Y 283.952,Z 764.457,A -85,B 0,C 180,E1 -16997.127,E2 -16997.127} C_VEL
LIN {X 0,Y 283.179,Z 768.27,A -85,B 0,C 180,E1 -16999.271,E2 -16999.271} C_VEL
LIN {X 0,Y 282.668,Z 771.063,A -85,B 0,C 180,E1 -17001.419,E2 -17001.419} C_VEL
LIN {X 0,Y 282.49,Z 772.371,A -85,B 0,C 180,E1 -17002.852,E2 -17002.852} C_VEL
LIN {X 0,Y 282.443,Z 773.337,A -85,B 0,C 180,E1 -17004.452,E2 -17004.452} C_VEL
LIN {X 0,Y 282.466,Z 773.73,A -85,B 0,C 180,E1 -17005.717,E2 -17005.717} C_VEL
LIN {X 0,Y 282.632,Z 774.056,A -85,B 0,C 180,E1 -17009.998,E2 -17009.998} C_VEL
LIN {X 0,Y 282.518,Z 773.292,A -85,B 0,C 180,E1 -17012.85,E2 -17012.85} C_VEL
LIN {X 0,Y 282.521,Z 771.055,A -85,B 0,C 180,E1 -17015.709,E2 -17015.709} C_VEL
LIN {X 0,Y 282.56,Z 768.411,A -85,B 0,C 180,E1 -17017.861,E2 -17017.861} C_VEL
LIN {X 0,Y 282.987,Z 763.411,A -85,B 0,C 180,E1 -17020.733,E2 -17020.733} C_VEL
LIN {X 0,Y 283.671,Z 758.559,A -85,B 0,C 180,E1 -17022.882,E2 -17022.882} C_VEL
LIN {X 0,Y 284.666,Z 751.138,A -85,B 0,C 180,E1 -17025.488,E2 -17025.488} C_VEL
LIN {X 0,Y 286.097,Z 744.005,A -85,B 0,C 180,E1 -17027.511,E2 -17027.511} C_VEL
LIN {X 0,Y 287.761,Z 734.995,A -85,B 0,C 180,E1 -17029.62,E2 -17029.62} C_VEL
LIN {X 0,Y 289.527,Z 726.033,A -85,B 0,C 180,E1 -17031.351,E2 -17031.351} C_VEL
LIN {X 0,Y 291.723,Z 714.101,A -85,B 0,C 180,E1 -17033.232,E2 -17033.232} C_VEL
LIN {X 0,Y 293.376,Z 704.031,A -85,B 0,C 180,E1 -17034.528,E2 -17034.528} C_VEL
LIN {X 0,Y 295.212,Z 692.313,A -85,B 0,C 180,E1 -17035.749,E2 -17035.749} C_VEL
LIN {X 0,Y 297.006,Z 679.215,A -85,B 0,C 180,E1 -17036.81,E2 -17036.81} C_VEL
LIN {X 0,Y 298.434,Z 665.799,A -85,B 0,C 180,E1 -17037.619,E2 -17037.619} C_VEL
LIN {X 0,Y 299.489,Z 652.188,A -85,B 0,C 180,E1 -17038.179,E2 -17038.179} C_VEL
LIN {X 0,Y 302.576,Z 562.132,A -85,B 0,C 180,E1 -17040.431,E2 -17040.431} C_VEL
LIN {X 0,Y 298.618,Z 532.59,A -85,B 0,C 180,E1 -17041.686,E2 -17041.686} C_VEL
LIN {X 0,Y 293.741,Z 521.224,A -85,B 0,C 180,E1 -17042.606,E2 -17042.606} C_VEL
LIN {X 0,Y 291.201,Z 510.418,A -85,B 0,C 180,E1 -17045.736,E2 -17045.736} C_VEL
LIN {X 0,Y 288.051,Z 498.822,A -85,B 0,C 180,E1 -17049.37,E2 -17049.37} C_VEL
LIN {X 0,Y 284.657,Z 487.934,A -85,B 0,C 180,E1 -17053.098,E2 -17053.098} C_VEL
LIN {X 0,Y 284.371,Z 486.686,A -85,B 0,C 180,E1 -17053.569,E2 -17053.569} C_VEL
LIN {X 0,Y 284.336,Z 486.685,A -85,B 0,C 180,E1 -17057.857,E2 -17057.857} C_VEL
LIN {X 0,Y 284.329,Z 486.687,A -85,B 0,C 180,E1 -17061.834,E2 -17061.834} C_VEL
LIN {X 0,Y 284.315,Z 486.67,A -85,B 0,C 180,E1 -17065.352,E2 -17065.352} C_VEL
LIN {X 0,Y 284.289,Z 486.689,A -85,B 0,C 180,E1 -17068.725,E2 -17068.725} C_VEL
LIN {X 0,Y 284.389,Z 486.679,A -85,B 0,C 180,E1 -17072.825,E2 -17072.825} C_VEL
LIN {X 0,Y 284.323,Z 486.661,A -85,B 0,C 180,E1 -17076.703,E2 -17076.703} C_VEL
LIN {X 0,Y 284.389,Z 486.684,A -85,B 0,C 180,E1 -17081.261,E2 -17081.261} C_VEL
LIN {X 0,Y 284.481,Z 486.664,A -85,B 0,C 180,E1 -17084.459,E2 -17084.459} C_VEL
LIN {X 0,Y 284.479,Z 486.664,A -85,B 0,C 180,E1 -17088.601,E2 -17088.601} C_VEL
LIN {X 0,Y 284.648,Z 486.652,A -85,B 0,C 180,E1 -17091.481,E2 -17091.481} C_VEL
LIN {X 0,Y 284.593,Z 486.648,A -85,B 0,C 180,E1 -17094.331,E2 -17094.331} C_VEL
LIN {X 0,Y 284.847,Z 486.616,A -85,B 0,C 180,E1 -17098.586,E2 -17098.586} C_VEL
LIN {X 0,Y 284.846,Z 486.627,A -85,B 0,C 180,E1 -17101.414,E2 -17101.414} C_VEL
LIN {X 0,Y 284.688,Z 486.643,A -85,B 0,C 180,E1 -17107.091,E2 -17107.091} C_VEL
LIN {X 0,Y 284.557,Z 486.66,A -85,B 0,C 180,E1 -17109.956,E2 -17109.956} C_VEL
LIN {X 0,Y 284.472,Z 486.667,A -85,B 0,C 180,E1 -17114.304,E2 -17114.304} C_VEL
LIN {X 0,Y 284.415,Z 486.673,A -85,B 0,C 180,E1 -17117.249,E2 -17117.249} C_VEL
LIN {X 0,Y 284.369,Z 486.689,A -85,B 0,C 180,E1 -17120.243,E2 -17120.243} C_VEL
LIN {X 0,Y 284.36,Z 486.687,A -85,B 0,C 180,E1 -17123.877,E2 -17123.877} C_VEL
LIN {X 0,Y 284.355,Z 486.688,A -85,B 0,C 180,E1 -17128.008,E2 -17128.008} C_VEL
LIN {X 0,Y 284.291,Z 486.694,A -85,B 0,C 180,E1 -17131.275,E2 -17131.275} C_VEL
LIN {X 0,Y 284.354,Z 486.69,A -85,B 0,C 180,E1 -17135.356,E2 -17135.356} C_VEL
LIN {X 0,Y 284.322,Z 486.691,A -85,B 0,C 180,E1 -17138.168,E2 -17138.168} C_VEL
LIN {X 0,Y 284.298,Z 486.7,A -85,B 0,C 180,E1 -17141.871,E2 -17141.871} C_VEL
LIN {X 0,Y 284.301,Z 486.693,A -85,B 0,C 180,E1 -17145.799,E2 -17145.799} C_VEL
LIN {X 0,Y 284.371,Z 486.831,A -85,B 0,C 180,E1 -17149.557,E2 -17149.557} C_VEL
LIN {X 0,Y 286.747,Z 495.217,A -85,B 0,C 180,E1 -17152.802,E2 -17152.802} C_VEL
LIN {X 0,Y 289.424,Z 505.451,A -85,B 0,C 180,E1 -17156.469,E2 -17156.469} C_VEL
LIN {X 0,Y 291.861,Z 516.417,A -85,B 0,C 180,E1 -17160.099,E2 -17160.099} C_VEL
LIN {X 0,Y 292.111,Z 517.602,A -85,B 0,C 180,E1 -17160.409,E2 -17160.409} C_VEL
LIN {X 0,Y 296.524,Z 527.688,A -85,B 0,C 180,E1 -17161.19,E2 -17161.19} C_VEL
LIN {X 0,Y 301.535,Z 553.548,A -85,B 0,C 180,E1 -17162.406,E2 -17162.406} C_VEL
LIN {X 0,Y 302.139,Z 557.755,A -85,B 0,C 180,E1 -17162.574,E2 -17162.574} C_VEL
LIN {X 0,Y 299.999,Z 633.847,A -85,B 0,C 180,E1 -17164.272,E2 -17164.272} C_VEL
LIN {X 0,Y 299.268,Z 646.594,A -85,B 0,C 180,E1 -17164.811,E2 -17164.811} C_VEL
LIN {X 0,Y 298.041,Z 659.677,A -85,B 0,C 180,E1 -17165.63,E2 -17165.63} C_VEL
LIN {X 0,Y 296.625,Z 671.256,A -85,B 0,C 180,E1 -17166.62,E2 -17166.62} C_VEL
LIN {X 0,Y 294.952,Z 681.859,A -85,B 0,C 180,E1 -17167.776,E2 -17167.776} C_VEL
LIN {X 0,Y 293.149,Z 692.384,A -85,B 0,C 180,E1 -17169.228,E2 -17169.228} C_VEL
LIN {X 0,Y 291.201,Z 702.532,A -85,B 0,C 180,E1 -17170.987,E2 -17170.987} C_VEL
LIN {X 0,Y 289.12,Z 712.04,A -85,B 0,C 180,E1 -17173.042,E2 -17173.042} C_VEL
LIN {X 0,Y 287.428,Z 719.714,A -85,B 0,C 180,E1 -17175.125,E2 -17175.125} C_VEL
LIN {X 0,Y 286.018,Z 725.909,A -85,B 0,C 180,E1 -17177.226,E2 -17177.226} C_VEL
LIN {X 0,Y 284.809,Z 730.883,A -85,B 0,C 180,E1 -17179.337,E2 -17179.337} C_VEL
LIN {X 0,Y 283.935,Z 734.779,A -85,B 0,C 180,E1 -17181.461,E2 -17181.461} C_VEL
LIN {X 0,Y 283.588,Z 736.853,A -85,B 0,C 180,E1 -17182.884,E2 -17182.884} C_VEL
LIN {X 0,Y 282.962,Z 739.767,A -85,B 0,C 180,E1 -17185.729,E2 -17185.729} C_VEL
LIN {X 0,Y 282.704,Z 741.229,A -85,B 0,C 180,E1 -17188.577,E2 -17188.577} C_VEL
LIN {X 0,Y 282.704,Z 741.264,A -85,B 0,C 180,E1 -17191.426,E2 -17191.426} C_VEL
LIN {X 0,Y 282.948,Z 739.848,A -85,B 0,C 180,E1 -17194.275,E2 -17194.275} C_VEL
LIN {X 0,Y 283.565,Z 736.986,A -85,B 0,C 180,E1 -17197.12,E2 -17197.12} C_VEL
LIN {X 0,Y 284.201,Z 733.772,A -85,B 0,C 180,E1 -17199.252,E2 -17199.252} C_VEL
LIN {X 0,Y 285.156,Z 729.571,A -85,B 0,C 180,E1 -17201.373,E2 -17201.373} C_VEL
LIN {X 0,Y 286.632,Z 723.293,A -85,B 0,C 180,E1 -17203.833,E2 -17203.833} C_VEL
LIN {X 0,Y 288.278,Z 716.479,A -85,B 0,C 180,E1 -17205.92,E2 -17205.92} C_VEL
LIN {X 0,Y 289.724,Z 709.589,A -85,B 0,C 180,E1 -17207.653,E2 -17207.653} C_VEL
LIN {X 0,Y 291.53,Z 701.323,A -85,B 0,C 180,E1 -17209.36,E2 -17209.36} C_VEL
LIN {X 0,Y 293.373,Z 691.231,A -85,B 0,C 180,E1 -17211.061,E2 -17211.061} C_VEL
LIN {X 0,Y 295.072,Z 681.313,A -85,B 0,C 180,E1 -17212.403,E2 -17212.403} C_VEL
LIN {X 0,Y 296.781,Z 670.573,A -85,B 0,C 180,E1 -17213.556,E2 -17213.556} C_VEL
LIN {X 0,Y 298.342,Z 657.671,A -85,B 0,C 180,E1 -17214.626,E2 -17214.626} C_VEL
LIN {X 0,Y 299.442,Z 644.613,A -85,B 0,C 180,E1 -17215.41,E2 -17215.41} C_VEL
LIN {X 0,Y 300.205,Z 631.682,A -85,B 0,C 180,E1 -17215.899,E2 -17215.899} C_VEL
LIN {X 0,Y 302.126,Z 556.546,A -85,B 0,C 180,E1 -17217.575,E2 -17217.575} C_VEL
LIN {X 0,Y 297.48,Z 532.02,A -85,B 0,C 180,E1 -17218.706,E2 -17218.706} C_VEL
LIN {X 0,Y 296.106,Z 526.511,A -85,B 0,C 180,E1 -17219.007,E2 -17219.007} C_VEL
LIN {X 0,Y 291.988,Z 517.273,A -85,B 0,C 180,E1 -17219.76,E2 -17219.76} C_VEL
LIN {X 0,Y 289.517,Z 505.851,A -85,B 0,C 180,E1 -17223.524,E2 -17223.524} C_VEL
LIN {X 0,Y 286.887,Z 495.454,A -85,B 0,C 180,E1 -17227.235,E2 -17227.235} C_VEL
LIN {X 0,Y 284.296,Z 486.693,A -85,B 0,C 180,E1 -17230.663,E2 -17230.663} C_VEL
LIN {X 0,Y 284.251,Z 486.694,A -85,B 0,C 180,E1 -17234.191,E2 -17234.191} C_VEL
LIN {X 0,Y 284.278,Z 486.688,A -85,B 0,C 180,E1 -17238.125,E2 -17238.125} C_VEL
LIN {X 0,Y 284.325,Z 486.679,A -85,B 0,C 180,E1 -17242.28,E2 -17242.28} C_VEL
LIN {X 0,Y 284.332,Z 486.688,A -85,B 0,C 180,E1 -17243.837,E2 -17243.837} C_VEL
LIN {X 0,Y 284.104,Z 487.207,A -85,B 0,C 180,E1 -17244.607,E2 -17244.607} C_VEL
LIN {X 0,Y 283.57,Z 488.543,A -85,B 0,C 180,E1 -17245.336,E2 -17245.336} C_VEL
LIN {X 0,Y 282.497,Z 491.601,A -85,B 0,C 180,E1 -17246.343,E2 -17246.343} C_VEL
LIN {X 0,Y 280.931,Z 498.433,A -85,B 0,C 180,E1 -17247.878,E2 -17247.878} C_VEL
LIN {X 0,Y 280.854,Z 502.737,A -85,B 0,C 180,E1 -17248.783,E2 -17248.783} C_VEL
LIN {X 0,Y 281.082,Z 504.108,A -85,B 0,C 180,E1 -17249.09,E2 -17249.09} C_VEL
LIN {X 0,Y 283.473,Z 515.032,A -85,B 0,C 180,E1 -17251.528,E2 -17251.528} C_VEL
LIN {X 0,Y 283.761,Z 518.918,A -85,B 0,C 180,E1 -17252.35,E2 -17252.35} C_VEL
LIN {X 0,Y 282.471,Z 534.307,A -85,B 0,C 180,E1 -17255.409,E2 -17255.409} C_VEL
LIN {X 0,Y 285.486,Z 561.87,A -85,B 0,C 180,E1 -17256.63,E2 -17256.63} C_VEL
LIN {X 0,Y 282.157,Z 646.163,A -85,B 0,C 180,E1 -17259.829,E2 -17259.829} C_VEL
LIN {X 0,Y 281.494,Z 659.347,A -85,B 0,C 180,E1 -17260.587,E2 -17260.587} C_VEL
LIN {X 0,Y 280.664,Z 673.845,A -85,B 0,C 180,E1 -17261.759,E2 -17261.759} C_VEL
LIN {X 0,Y 279.617,Z 686.616,A -85,B 0,C 180,E1 -17263.13,E2 -17263.13} C_VEL
LIN {X 0,Y 278.795,Z 696.624,A -85,B 0,C 180,E1 -17264.464,E2 -17264.464} C_VEL
LIN {X 0,Y 277.951,Z 706.729,A -85,B 0,C 180,E1 -17266.101,E2 -17266.101} C_VEL
LIN {X 0,Y 277.03,Z 717.643,A -85,B 0,C 180,E1 -17268.29,E2 -17268.29} C_VEL
LIN {X 0,Y 276.341,Z 726.329,A -85,B 0,C 180,E1 -17270.485,E2 -17270.485} C_VEL
LIN {X 0,Y 275.849,Z 733.341,A -85,B 0,C 180,E1 -17272.681,E2 -17272.681} C_VEL
LIN {X 0,Y 275.539,Z 739.295,A -85,B 0,C 180,E1 -17275.074,E2 -17275.074} C_VEL
LIN {X 0,Y 275.48,Z 743.166,A -85,B 0,C 180,E1 -17277.075,E2 -17277.075} C_VEL
LIN {X 0,Y 275.385,Z 745.38,A -85,B 0,C 180,E1 -17278.537,E2 -17278.537} C_VEL
LIN {X 0,Y 275.38,Z 747.169,A -85,B 0,C 180,E1 -17280,E2 -17280} C_VEL
LIN {X 0,Y 275.504,Z 748.48,A -85,B 0,C 180,E1 -17281.462,E2 -17281.462} C_VEL
LIN {X 0,Y 275.696,Z 749.348,A -85,B 0,C 180,E1 -17282.922,E2 -17282.922} C_VEL
LIN {X 0,Y 275.904,Z 749.808,A -85,B 0,C 180,E1 -17284.382,E2 -17284.382} C_VEL
LIN {X 0,Y 276.208,Z 749.842,A -85,B 0,C 180,E1 -17285.841,E2 -17285.841} C_VEL
LIN {X 0,Y 276.711,Z 749.414,A -85,B 0,C 180,E1 -17287.296,E2 -17287.296} C_VEL
LIN {X 0,Y 277.377,Z 748.531,A -85,B 0,C 180,E1 -17288.818,E2 -17288.818} C_VEL
LIN {X 0,Y 278.064,Z 747.338,A -85,B 0,C 180,E1 -17290.19,E2 -17290.19} C_VEL
LIN {X 0,Y 279.38,Z 744.627,A -85,B 0,C 180,E1 -17292.346,E2 -17292.346} C_VEL
LIN {X 0,Y 281.12,Z 740.88,A -85,B 0,C 180,E1 -17294.477,E2 -17294.477} C_VEL
LIN {X 0,Y 283.083,Z 735.993,A -85,B 0,C 180,E1 -17296.589,E2 -17296.589} C_VEL
LIN {X 0,Y 285.911,Z 728.679,A -85,B 0,C 180,E1 -17299.008,E2 -17299.008} C_VEL
LIN {X 0,Y 288.785,Z 720.822,A -85,B 0,C 180,E1 -17301.036,E2 -17301.036} C_VEL
LIN {X 0,Y 292.022,Z 711.021,A -85,B 0,C 180,E1 -17303.022,E2 -17303.022} C_VEL
LIN {X 0,Y 295.044,Z 700.776,A -85,B 0,C 180,E1 -17304.707,E2 -17304.707} C_VEL
LIN {X 0,Y 298.095,Z 689.029,A -85,B 0,C 180,E1 -17306.235,E2 -17306.235} C_VEL
LIN {X 0,Y 300.8,Z 677.092,A -85,B 0,C 180,E1 -17307.443,E2 -17307.443} C_VEL
LIN {X 0,Y 303.242,Z 664.327,A -85,B 0,C 180,E1 -17308.461,E2 -17308.461} C_VEL
LIN {X 0,Y 305.355,Z 650.167,A -85,B 0,C 180,E1 -17309.28,E2 -17309.28} C_VEL
LIN {X 0,Y 314.495,Z 581.803,A -85,B 0,C 180,E1 -17312.178,E2 -17312.178} C_VEL
LIN {X 0,Y 315.372,Z 575.077,A -85,B 0,C 180,E1 -17312.495,E2 -17312.495} C_VEL
LIN {X 0,Y 314.472,Z 563.212,A -85,B 0,C 180,E1 -17313.903,E2 -17313.903} C_VEL
LIN {X 0,Y 314.002,Z 558.946,A -85,B 0,C 180,E1 -17314.517,E2 -17314.517} C_VEL
LIN {X 0,Y 311.744,Z 552.727,A -85,B 0,C 180,E1 -17316.208,E2 -17316.208} C_VEL
LIN {X 0,Y 309.692,Z 547.76,A -85,B 0,C 180,E1 -17318.048,E2 -17318.048} C_VEL
LIN {X 0,Y 308.045,Z 543.609,A -85,B 0,C 180,E1 -17320.159,E2 -17320.159} C_VEL
LIN {X 0,Y 308.07,Z 542.241,A -85,B 0,C 180,E1 -17321.42,E2 -17321.42} C_VEL
LIN {X 0,Y 308.235,Z 540.934,A -85,B 0,C 180,E1 -17323.159,E2 -17323.159} C_VEL
LIN {X 0,Y 308.648,Z 540.26,A -85,B 0,C 180,E1 -17325.098,E2 -17325.098} C_VEL
LIN {X 0,Y 309.359,Z 540.413,A -85,B 0,C 180,E1 -17327.034,E2 -17327.034} C_VEL
LIN {X 0,Y 310.479,Z 541.263,A -85,B 0,C 180,E1 -17328.969,E2 -17328.969} C_VEL
LIN {X 0,Y 312.069,Z 542.971,A -85,B 0,C 180,E1 -17330.905,E2 -17330.905} C_VEL
LIN {X 0,Y 312.354,Z 544.007,A -85,B 0,C 180,E1 -17331.447,E2 -17331.447} C_VEL
LIN {X 0,Y 312.536,Z 549.22,A -85,B 0,C 180,E1 -17332.968,E2 -17332.968} C_VEL
LIN {X 0,Y 314.022,Z 555.353,A -85,B 0,C 180,E1 -17334.364,E2 -17334.364} C_VEL
LIN {X 0,Y 313.901,Z 561.065,A -85,B 0,C 180,E1 -17334.92,E2 -17334.92} C_VEL
LIN {X 0,Y 313.553,Z 568.116,A -85,B 0,C 180,E1 -17335.491,E2 -17335.491} C_VEL
LIN {X 0,Y 300.564,Z 659.165,A -85,B 0,C 180,E1 -17339.478,E2 -17339.478} C_VEL
LIN {X 0,Y 298.521,Z 674.482,A -85,B 0,C 180,E1 -17340.271,E2 -17340.271} C_VEL
LIN {X 0,Y 296.088,Z 688.648,A -85,B 0,C 180,E1 -17341.27,E2 -17341.27} C_VEL
LIN {X 0,Y 293.71,Z 700.497,A -85,B 0,C 180,E1 -17342.377,E2 -17342.377} C_VEL
LIN {X 0,Y 290.914,Z 712.805,A -85,B 0,C 180,E1 -17343.815,E2 -17343.815} C_VEL
LIN {X 0,Y 288.207,Z 724.175,A -85,B 0,C 180,E1 -17345.507,E2 -17345.507} C_VEL
LIN {X 0,Y 285.595,Z 733.688,A -85,B 0,C 180,E1 -17347.194,E2 -17347.194} C_VEL
LIN {X 0,Y 282.972,Z 743.147,A -85,B 0,C 180,E1 -17349.271,E2 -17349.271} C_VEL
LIN {X 0,Y 280.779,Z 750.961,A -85,B 0,C 180,E1 -17351.388,E2 -17351.388} C_VEL
LIN {X 0,Y 278.748,Z 758.33,A -85,B 0,C 180,E1 -17353.897,E2 -17353.897} C_VEL
LIN {X 0,Y 277.448,Z 763.374,A -85,B 0,C 180,E1 -17356.074,E2 -17356.074} C_VEL
LIN {X 0,Y 276.41,Z 767.309,A -85,B 0,C 180,E1 -17358.262,E2 -17358.262} C_VEL
LIN {X 0,Y 275.965,Z 769.399,A -85,B 0,C 180,E1 -17359.729,E2 -17359.729} C_VEL
LIN {X 0,Y 275.619,Z 771.011,A -85,B 0,C 180,E1 -17361.198,E2 -17361.198} C_VEL
LIN {X 0,Y 275.416,Z 772.213,A -85,B 0,C 180,E1 -17362.668,E2 -17362.668} C_VEL
LIN {X 0,Y 275.355,Z 773.137,A -85,B 0,C 180,E1 -17364.511,E2 -17364.511} C_VEL
LIN {X 0,Y 275.469,Z 773.456,A -85,B 0,C 180,E1 -17368.536,E2 -17368.536} C_VEL
LIN {X 0,Y 275.542,Z 773.647,A -85,B 0,C 180,E1 -17369.998,E2 -17369.998} C_VEL
LIN {X 0,Y 275.443,Z 772.883,A -85,B 0,C 180,E1 -17372.923,E2 -17372.923} C_VEL
LIN {X 0,Y 275.444,Z 770.642,A -85,B 0,C 180,E1 -17375.856,E2 -17375.856} C_VEL
LIN {X 0,Y 275.577,Z 766.879,A -85,B 0,C 180,E1 -17378.8,E2 -17378.8} C_VEL
LIN {X 0,Y 276.127,Z 761.503,A -85,B 0,C 180,E1 -17381.746,E2 -17381.746} C_VEL
LIN {X 0,Y 276.966,Z 756.255,A -85,B 0,C 180,E1 -17383.947,E2 -17383.947} C_VEL
LIN {X 0,Y 278.025,Z 749.872,A -85,B 0,C 180,E1 -17386.142,E2 -17386.142} C_VEL
LIN {X 0,Y 279.511,Z 742.171,A -85,B 0,C 180,E1 -17388.316,E2 -17388.316} C_VEL
LIN {X 0,Y 281.33,Z 732.876,A -85,B 0,C 180,E1 -17390.469,E2 -17390.469} C_VEL
LIN {X 0,Y 283.494,Z 722.584,A -85,B 0,C 180,E1 -17392.403,E2 -17392.403} C_VEL
LIN {X 0,Y 285.627,Z 711.01,A -85,B 0,C 180,E1 -17394.167,E2 -17394.167} C_VEL
LIN {X 0,Y 287.502,Z 700.056,A -85,B 0,C 180,E1 -17395.518,E2 -17395.518} C_VEL
LIN {X 0,Y 289.358,Z 688.068,A -85,B 0,C 180,E1 -17396.699,E2 -17396.699} C_VEL
LIN {X 0,Y 291.08,Z 674.904,A -85,B 0,C 180,E1 -17397.694,E2 -17397.694} C_VEL
LIN {X 0,Y 292.513,Z 661.521,A -85,B 0,C 180,E1 -17398.424,E2 -17398.424} C_VEL
LIN {X 0,Y 293.369,Z 648.115,A -85,B 0,C 180,E1 -17398.919,E2 -17398.919} C_VEL
LIN {X 0,Y 296.29,Z 562.152,A -85,B 0,C 180,E1 -17401.102,E2 -17401.102} C_VEL
LIN {X 0,Y 292.59,Z 534.848,A -85,B 0,C 180,E1 -17402.306,E2 -17402.306} C_VEL
LIN {X 0,Y 286.571,Z 521.182,A -85,B 0,C 180,E1 -17403.462,E2 -17403.462} C_VEL
LIN {X 0,Y 284.279,Z 511.435,A -85,B 0,C 180,E1 -17406.391,E2 -17406.391} C_VEL
LIN {X 0,Y 281.422,Z 500.909,A -85,B 0,C 180,E1 -17409.807,E2 -17409.807} C_VEL
LIN {X 0,Y 278.252,Z 490.629,A -85,B 0,C 180,E1 -17413.44,E2 -17413.44} C_VEL
LIN {X 0,Y 277.307,Z 487.568,A -85,B 0,C 180,E1 -17414.603,E2 -17414.603} C_VEL
LIN {X 0,Y 277.286,Z 487.567,A -85,B 0,C 180,E1 -17418.778,E2 -17418.778} C_VEL
LIN {X 0,Y 277.282,Z 487.552,A -85,B 0,C 180,E1 -17422.533,E2 -17422.533} C_VEL
LIN {X 0,Y 277.245,Z 487.562,A -85,B 0,C 180,E1 -17426.104,E2 -17426.104} C_VEL
LIN {X 0,Y 277.252,Z 487.569,A -85,B 0,C 180,E1 -17429.538,E2 -17429.538} C_VEL
LIN {X 0,Y 277.351,Z 487.556,A -85,B 0,C 180,E1 -17432.863,E2 -17432.863} C_VEL
LIN {X 0,Y 277.287,Z 487.547,A -85,B 0,C 180,E1 -17436.076,E2 -17436.076} C_VEL
LIN {X 0,Y 277.332,Z 487.556,A -85,B 0,C 180,E1 -17440.765,E2 -17440.765} C_VEL
LIN {X 0,Y 277.424,Z 487.549,A -85,B 0,C 180,E1 -17445.326,E2 -17445.326} C_VEL
LIN {X 0,Y 277.496,Z 487.538,A -85,B 0,C 180,E1 -17449.789,E2 -17449.789} C_VEL
LIN {X 0,Y 277.643,Z 487.515,A -85,B 0,C 180,E1 -17452.729,E2 -17452.729} C_VEL
LIN {X 0,Y 277.812,Z 487.492,A -85,B 0,C 180,E1 -17458.551,E2 -17458.551} C_VEL
LIN {X 0,Y 277.812,Z 487.503,A -85,B 0,C 180,E1 -17461.45,E2 -17461.45} C_VEL
LIN {X 0,Y 277.642,Z 487.52,A -85,B 0,C 180,E1 -17467.271,E2 -17467.271} C_VEL
LIN {X 0,Y 277.497,Z 487.541,A -85,B 0,C 180,E1 -17470.212,E2 -17470.212} C_VEL
LIN {X 0,Y 277.425,Z 487.548,A -85,B 0,C 180,E1 -17474.675,E2 -17474.675} C_VEL
LIN {X 0,Y 277.335,Z 487.562,A -85,B 0,C 180,E1 -17479.235,E2 -17479.235} C_VEL
LIN {X 0,Y 277.31,Z 487.567,A -85,B 0,C 180,E1 -17484.172,E2 -17484.172} C_VEL
LIN {X 0,Y 277.326,Z 487.562,A -85,B 0,C 180,E1 -17487.51,E2 -17487.51} C_VEL
LIN {X 0,Y 277.263,Z 487.565,A -85,B 0,C 180,E1 -17490.483,E2 -17490.483} C_VEL
LIN {X 0,Y 277.247,Z 487.567,A -85,B 0,C 180,E1 -17493.896,E2 -17493.896} C_VEL
LIN {X 0,Y 277.278,Z 487.565,A -85,B 0,C 180,E1 -17497.468,E2 -17497.468} C_VEL
LIN {X 0,Y 277.235,Z 487.577,A -85,B 0,C 180,E1 -17501.232,E2 -17501.232} C_VEL
LIN {X 0,Y 277.244,Z 487.574,A -85,B 0,C 180,E1 -17505.218,E2 -17505.218} C_VEL
LIN {X 0,Y 277.322,Z 487.687,A -85,B 0,C 180,E1 -17508.545,E2 -17508.545} C_VEL
LIN {X 0,Y 279.913,Z 496.656,A -85,B 0,C 180,E1 -17512.148,E2 -17512.148} C_VEL
LIN {X 0,Y 282.377,Z 506.183,A -85,B 0,C 180,E1 -17515.673,E2 -17515.673} C_VEL
LIN {X 0,Y 284.97,Z 517.491,A -85,B 0,C 180,E1 -17519.531,E2 -17519.531} C_VEL
LIN {X 0,Y 290.668,Z 530.181,A -85,B 0,C 180,E1 -17520.577,E2 -17520.577} C_VEL
LIN {X 0,Y 295.473,Z 555.393,A -85,B 0,C 180,E1 -17521.795,E2 -17521.795} C_VEL
LIN {X 0,Y 295.925,Z 557.957,A -85,B 0,C 180,E1 -17521.91,E2 -17521.91} C_VEL
LIN {X 0,Y 293.734,Z 633.729,A -85,B 0,C 180,E1 -17523.634,E2 -17523.634} C_VEL
LIN {X 0,Y 292.959,Z 646.604,A -85,B 0,C 180,E1 -17524.181,E2 -17524.181} C_VEL
LIN {X 0,Y 291.629,Z 660.322,A -85,B 0,C 180,E1 -17525.058,E2 -17525.058} C_VEL
LIN {X 0,Y 290.148,Z 671.823,A -85,B 0,C 180,E1 -17526.066,E2 -17526.066} C_VEL
LIN {X 0,Y 288.43,Z 682.375,A -85,B 0,C 180,E1 -17527.246,E2 -17527.246} C_VEL
LIN {X 0,Y 286.444,Z 693.336,A -85,B 0,C 180,E1 -17528.804,E2 -17528.804} C_VEL
LIN {X 0,Y 284.528,Z 702.983,A -85,B 0,C 180,E1 -17530.523,E2 -17530.523} C_VEL
LIN {X 0,Y 282.363,Z 712.477,A -85,B 0,C 180,E1 -17532.624,E2 -17532.624} C_VEL
LIN {X 0,Y 280.585,Z 720.142,A -85,B 0,C 180,E1 -17534.754,E2 -17534.754} C_VEL
LIN {X 0,Y 279.12,Z 726.329,A -85,B 0,C 180,E1 -17536.904,E2 -17536.904} C_VEL
LIN {X 0,Y 277.849,Z 731.3,A -85,B 0,C 180,E1 -17539.066,E2 -17539.066} C_VEL
LIN {X 0,Y 276.931,Z 735.192,A -85,B 0,C 180,E1 -17541.244,E2 -17541.244} C_VEL
LIN {X 0,Y 276.541,Z 737.265,A -85,B 0,C 180,E1 -17542.702,E2 -17542.702} C_VEL
LIN {X 0,Y 275.904,Z 740.176,A -85,B 0,C 180,E1 -17545.619,E2 -17545.619} C_VEL
LIN {X 0,Y 275.618,Z 741.639,A -85,B 0,C 180,E1 -17548.541,E2 -17548.541} C_VEL
LIN {X 0,Y 275.618,Z 741.673,A -85,B 0,C 180,E1 -17551.463,E2 -17551.463} C_VEL
LIN {X 0,Y 275.891,Z 740.257,A -85,B 0,C 180,E1 -17554.385,E2 -17554.385} C_VEL
LIN {X 0,Y 276.524,Z 737.396,A -85,B 0,C 180,E1 -17557.303,E2 -17557.303} C_VEL
LIN {X 0,Y 277.201,Z 734.183,A -85,B 0,C 180,E1 -17559.487,E2 -17559.487} C_VEL
LIN {X 0,Y 278.2,Z 729.986,A -85,B 0,C 180,E1 -17561.662,E2 -17561.662} C_VEL
LIN {X 0,Y 279.754,Z 723.711,A -85,B 0,C 180,E1 -17564.18,E2 -17564.18} C_VEL
LIN {X 0,Y 281.468,Z 716.905,A -85,B 0,C 180,E1 -17566.316,E2 -17566.316} C_VEL
LIN {X 0,Y 283.003,Z 710.02,A -85,B 0,C 180,E1 -17568.086,E2 -17568.086} C_VEL
LIN {X 0,Y 284.869,Z 701.768,A -85,B 0,C 180,E1 -17569.831,E2 -17569.831} C_VEL
LIN {X 0,Y 286.785,Z 691.707,A -85,B 0,C 180,E1 -17571.569,E2 -17571.569} C_VEL
LIN {X 0,Y 288.822,Z 680.406,A -85,B 0,C 180,E1 -17573.104,E2 -17573.104} C_VEL
LIN {X 0,Y 290.563,Z 669.37,A -85,B 0,C 180,E1 -17574.281,E2 -17574.281} C_VEL
LIN {X 0,Y 292.058,Z 657.169,A -85,B 0,C 180,E1 -17575.287,E2 -17575.287} C_VEL
LIN {X 0,Y 293.133,Z 644.571,A -85,B 0,C 180,E1 -17576.045,E2 -17576.045} C_VEL
LIN {X 0,Y 293.934,Z 631.398,A -85,B 0,C 180,E1 -17576.542,E2 -17576.542} C_VEL
LIN {X 0,Y 295.886,Z 557.411,A -85,B 0,C 180,E1 -17578.228,E2 -17578.228} C_VEL
LIN {X 0,Y 291.222,Z 532.676,A -85,B 0,C 180,E1 -17579.41,E2 -17579.41} C_VEL
LIN {X 0,Y 290.043,Z 528.729,A -85,B 0,C 180,E1 -17579.658,E2 -17579.658} C_VEL
LIN {X 0,Y 284.888,Z 517.369,A -85,B 0,C 180,E1 -17580.619,E2 -17580.619} C_VEL
LIN {X 0,Y 282.712,Z 507.609,A -85,B 0,C 180,E1 -17583.95,E2 -17583.95} C_VEL
LIN {X 0,Y 280.41,Z 498.298,A -85,B 0,C 180,E1 -17587.343,E2 -17587.343} C_VEL
LIN {X 0,Y 277.936,Z 489.986,A -85,B 0,C 180,E1 -17590.659,E2 -17590.659} C_VEL
LIN {X 0,Y 277.239,Z 487.571,A -85,B 0,C 180,E1 -17591.718,E2 -17591.718} C_VEL
LIN {X 0,Y 277.208,Z 487.575,A -85,B 0,C 180,E1 -17595.227,E2 -17595.227} C_VEL
LIN {X 0,Y 277.229,Z 487.577,A -85,B 0,C 180,E1 -17599.513,E2 -17599.513} C_VEL
LIN {X 0,Y 277.271,Z 487.558,A -85,B 0,C 180,E1 -17602.531,E2 -17602.531} C_VEL
LIN {X 0,Y 277.321,Z 487.589,A -85,B 0,C 180,E1 -17605.295,E2 -17605.295} C_VEL
LIN {X 0,Y 281.082,Z 504.108,A -85,B 0,C 180,E1 -17609.09,E2 -17609.09} C_VEL
LIN {X 0,Y 281.262,Z 508.196,A -85,B 0,C 180,E1 -17609.963,E2 -17609.963} C_VEL
LIN {X 0,Y 280.404,Z 512.457,A -85,B 0,C 180,E1 -17610.795,E2 -17610.795} C_VEL
LIN {X 0,Y 276.675,Z 524.035,A -85,B 0,C 180,E1 -17612.986,E2 -17612.986} C_VEL
LIN {X 0,Y 276.201,Z 526.931,A -85,B 0,C 180,E1 -17613.564,E2 -17613.564} C_VEL
LIN {X 0,Y 275.546,Z 534.482,A -85,B 0,C 180,E1 -17615.077,E2 -17615.077} C_VEL
LIN {X 0,Y 278.478,Z 563.15,A -85,B 0,C 180,E1 -17616.384,E2 -17616.384} C_VEL
LIN {X 0,Y 275.076,Z 647.65,A -85,B 0,C 180,E1 -17619.726,E2 -17619.726} C_VEL
LIN {X 0,Y 274.361,Z 661.03,A -85,B 0,C 180,E1 -17620.548,E2 -17620.548} C_VEL
LIN {X 0,Y 273.588,Z 674.234,A -85,B 0,C 180,E1 -17621.658,E2 -17621.658} C_VEL
LIN {X 0,Y 272.532,Z 686.969,A -85,B 0,C 180,E1 -17623.061,E2 -17623.061} C_VEL
LIN {X 0,Y 271.679,Z 697,A -85,B 0,C 180,E1 -17624.431,E2 -17624.431} C_VEL
LIN {X 0,Y 270.813,Z 707.106,A -85,B 0,C 180,E1 -17626.11,E2 -17626.11} C_VEL
LIN {X 0,Y 269.907,Z 717.98,A -85,B 0,C 180,E1 -17628.358,E2 -17628.358} C_VEL
LIN {X 0,Y 269.228,Z 726.64,A -85,B 0,C 180,E1 -17630.61,E2 -17630.61} C_VEL
LIN {X 0,Y 268.723,Z 733.744,A -85,B 0,C 180,E1 -17632.901,E2 -17632.901} C_VEL
LIN {X 0,Y 268.472,Z 738.125,A -85,B 0,C 180,E1 -17634.646,E2 -17634.646} C_VEL
LIN {X 0,Y 268.389,Z 742.882,A -85,B 0,C 180,E1 -17636.998,E2 -17636.998} C_VEL
LIN {X 0,Y 268.31,Z 745.252,A -85,B 0,C 180,E1 -17638.499,E2 -17638.499} C_VEL
LIN {X 0,Y 268.3,Z 747.135,A -85,B 0,C 180,E1 -17640,E2 -17640} C_VEL
LIN {X 0,Y 268.425,Z 748.581,A -85,B 0,C 180,E1 -17641.5,E2 -17641.5} C_VEL
LIN {X 0,Y 268.624,Z 749.579,A -85,B 0,C 180,E1 -17642.999,E2 -17642.999} C_VEL
LIN {X 0,Y 268.85,Z 750.137,A -85,B 0,C 180,E1 -17644.498,E2 -17644.498} C_VEL
LIN {X 0,Y 269.161,Z 750.294,A -85,B 0,C 180,E1 -17645.995,E2 -17645.995} C_VEL
LIN {X 0,Y 269.718,Z 750.027,A -85,B 0,C 180,E1 -17647.486,E2 -17647.486} C_VEL
LIN {X 0,Y 271.13,Z 748.18,A -85,B 0,C 180,E1 -17650.454,E2 -17650.454} C_VEL
LIN {X 0,Y 272.526,Z 745.695,A -85,B 0,C 180,E1 -17652.662,E2 -17652.662} C_VEL
LIN {X 0,Y 274.362,Z 742.156,A -85,B 0,C 180,E1 -17654.842,E2 -17654.842} C_VEL
LIN {X 0,Y 276.468,Z 737.567,A -85,B 0,C 180,E1 -17656.998,E2 -17656.998} C_VEL
LIN {X 0,Y 279.033,Z 731.742,A -85,B 0,C 180,E1 -17659.113,E2 -17659.113} C_VEL
LIN {X 0,Y 281.416,Z 725.791,A -85,B 0,C 180,E1 -17660.847,E2 -17660.847} C_VEL
LIN {X 0,Y 284.701,Z 717.224,A -85,B 0,C 180,E1 -17662.88,E2 -17662.88} C_VEL
LIN {X 0,Y 288.282,Z 706.678,A -85,B 0,C 180,E1 -17664.855,E2 -17664.855} C_VEL
LIN {X 0,Y 291.734,Z 695.139,A -85,B 0,C 180,E1 -17666.555,E2 -17666.555} C_VEL
LIN {X 0,Y 294.722,Z 683.667,A -85,B 0,C 180,E1 -17667.903,E2 -17667.903} C_VEL
LIN {X 0,Y 297.543,Z 671.084,A -85,B 0,C 180,E1 -17669.038,E2 -17669.038} C_VEL
LIN {X 0,Y 299.951,Z 657.838,A -85,B 0,C 180,E1 -17669.958,E2 -17669.958} C_VEL
LIN {X 0,Y 302.154,Z 642.649,A -85,B 0,C 180,E1 -17670.695,E2 -17670.695} C_VEL
LIN {X 0,Y 311.638,Z 577.613,A -85,B 0,C 180,E1 -17673.504,E2 -17673.504} C_VEL
LIN {X 0,Y 311.023,Z 565.63,A -85,B 0,C 180,E1 -17674.995,E2 -17674.995} C_VEL
LIN {X 0,Y 310.735,Z 563.476,A -85,B 0,C 180,E1 -17675.37,E2 -17675.37} C_VEL
LIN {X 0,Y 308.953,Z 558.187,A -85,B 0,C 180,E1 -17676.917,E2 -17676.917} C_VEL
LIN {X 0,Y 307.384,Z 553.956,A -85,B 0,C 180,E1 -17678.532,E2 -17678.532} C_VEL
LIN {X 0,Y 305.88,Z 549.885,A -85,B 0,C 180,E1 -17680.691,E2 -17680.691} C_VEL
LIN {X 0,Y 305.008,Z 547.183,A -85,B 0,C 180,E1 -17683.316,E2 -17683.316} C_VEL
LIN {X 0,Y 305.144,Z 546.357,A -85,B 0,C 180,E1 -17685.56,E2 -17685.56} C_VEL
LIN {X 0,Y 305.824,Z 546.6,A -85,B 0,C 180,E1 -17687.339,E2 -17687.339} C_VEL
LIN {X 0,Y 307.263,Z 547.749,A -85,B 0,C 180,E1 -17689.34,E2 -17689.34} C_VEL
LIN {X 0,Y 308.781,Z 549.5,A -85,B 0,C 180,E1 -17690.882,E2 -17690.882} C_VEL
LIN {X 0,Y 309.981,Z 555.514,A -85,B 0,C 180,E1 -17692.517,E2 -17692.517} C_VEL
LIN {X 0,Y 310.873,Z 560.012,A -85,B 0,C 180,E1 -17693.529,E2 -17693.529} C_VEL
LIN {X 0,Y 310.255,Z 569.563,A -85,B 0,C 180,E1 -17694.359,E2 -17694.359} C_VEL
LIN {X 0,Y 296.552,Z 658.647,A -85,B 0,C 180,E1 -17698.324,E2 -17698.324} C_VEL
LIN {X 0,Y 294.149,Z 674.911,A -85,B 0,C 180,E1 -17699.188,E2 -17699.188} C_VEL
LIN {X 0,Y 291.416,Z 689.206,A -85,B 0,C 180,E1 -17700.229,E2 -17700.229} C_VEL
LIN {X 0,Y 288.471,Z 702.152,A -85,B 0,C 180,E1 -17701.49,E2 -17701.49} C_VEL
LIN {X 0,Y 285.541,Z 713.76,A -85,B 0,C 180,E1 -17702.908,E2 -17702.908} C_VEL
LIN {X 0,Y 282.09,Z 726.668,A -85,B 0,C 180,E1 -17704.94,E2 -17704.94} C_VEL
LIN {X 0,Y 279.282,Z 735.624,A -85,B 0,C 180,E1 -17706.649,E2 -17706.649} C_VEL
LIN {X 0,Y 276.48,Z 744.588,A -85,B 0,C 180,E1 -17708.761,E2 -17708.761} C_VEL
LIN {X 0,Y 274.145,Z 752.008,A -85,B 0,C 180,E1 -17710.92,E2 -17710.92} C_VEL
LIN {X 0,Y 271.961,Z 759.048,A -85,B 0,C 180,E1 -17713.483,E2 -17713.483} C_VEL
LIN {X 0,Y 270.562,Z 763.802,A -85,B 0,C 180,E1 -17715.712,E2 -17715.712} C_VEL
LIN {X 0,Y 269.421,Z 767.541,A -85,B 0,C 180,E1 -17717.953,E2 -17717.953} C_VEL
LIN {X 0,Y 268.933,Z 769.454,A -85,B 0,C 180,E1 -17719.458,E2 -17719.458} C_VEL
LIN {X 0,Y 268.335,Z 772.065,A -85,B 0,C 180,E1 -17722.473,E2 -17722.473} C_VEL
LIN {X 0,Y 268.26,Z 772.857,A -85,B 0,C 180,E1 -17724.586,E2 -17724.586} C_VEL
LIN {X 0,Y 268.355,Z 772.754,A -85,B 0,C 180,E1 -17726.996,E2 -17726.996} C_VEL
LIN {X 0,Y 268.454,Z 773.238,A -85,B 0,C 180,E1 -17729.998,E2 -17729.998} C_VEL
LIN {X 0,Y 268.368,Z 772.473,A -85,B 0,C 180,E1 -17733,E2 -17733} C_VEL
LIN {X 0,Y 268.35,Z 770.229,A -85,B 0,C 180,E1 -17736.011,E2 -17736.011} C_VEL
LIN {X 0,Y 268.5,Z 766.462,A -85,B 0,C 180,E1 -17739.034,E2 -17739.034} C_VEL
LIN {X 0,Y 269.123,Z 761.084,A -85,B 0,C 180,E1 -17742.057,E2 -17742.057} C_VEL
LIN {X 0,Y 270.176,Z 754.873,A -85,B 0,C 180,E1 -17744.69,E2 -17744.69} C_VEL
LIN {X 0,Y 271.146,Z 749.441,A -85,B 0,C 180,E1 -17746.564,E2 -17746.564} C_VEL
LIN {X 0,Y 272.721,Z 741.732,A -85,B 0,C 180,E1 -17748.789,E2 -17748.789} C_VEL
LIN {X 0,Y 274.614,Z 732.424,A -85,B 0,C 180,E1 -17750.993,E2 -17750.993} C_VEL
LIN {X 0,Y 276.856,Z 722.113,A -85,B 0,C 180,E1 -17752.971,E2 -17752.971} C_VEL
LIN {X 0,Y 278.984,Z 711.297,A -85,B 0,C 180,E1 -17754.66,E2 -17754.66} C_VEL
LIN {X 0,Y 281.079,Z 699.508,A -85,B 0,C 180,E1 -17756.145,E2 -17756.145} C_VEL
LIN {X 0,Y 283.02,Z 687.467,A -85,B 0,C 180,E1 -17757.346,E2 -17757.346} C_VEL
LIN {X 0,Y 284.801,Z 674.208,A -85,B 0,C 180,E1 -17758.359,E2 -17758.359} C_VEL
LIN {X 0,Y 286.304,Z 659.752,A -85,B 0,C 180,E1 -17759.148,E2 -17759.148} C_VEL
LIN {X 0,Y 287.249,Z 645.422,A -85,B 0,C 180,E1 -17759.646,E2 -17759.646} C_VEL
LIN {X 0,Y 290.116,Z 563.097,A -85,B 0,C 180,E1 -17761.766,E2 -17761.766} C_VEL
LIN {X 0,Y 286.742,Z 537.589,A -85,B 0,C 180,E1 -17762.919,E2 -17762.919} C_VEL
LIN {X 0,Y 279.458,Z 521.203,A -85,B 0,C 180,E1 -17764.351,E2 -17764.351} C_VEL
LIN {X 0,Y 276.982,Z 511.169,A -85,B 0,C 180,E1 -17767.512,E2 -17767.512} C_VEL
LIN {X 0,Y 274.244,Z 501.25,A -85,B 0,C 180,E1 -17770.888,E2 -17770.888} C_VEL
LIN {X 0,Y 271.249,Z 491.801,A -85,B 0,C 180,E1 -17774.389,E2 -17774.389} C_VEL
LIN {X 0,Y 270.214,Z 488.447,A -85,B 0,C 180,E1 -17775.761,E2 -17775.761} C_VEL
LIN {X 0,Y 270.241,Z 488.441,A -85,B 0,C 180,E1 -17779.446,E2 -17779.446} C_VEL
LIN {X 0,Y 270.249,Z 488.414,A -85,B 0,C 180,E1 -17783.72,E2 -17783.72} C_VEL
LIN {X 0,Y 270.196,Z 488.449,A -85,B 0,C 180,E1 -17786.892,E2 -17786.892} C_VEL
LIN {X 0,Y 270.22,Z 488.45,A -85,B 0,C 180,E1 -17790.386,E2 -17790.386} C_VEL
LIN {X 0,Y 270.254,Z 488.446,A -85,B 0,C 180,E1 -17793.763,E2 -17793.763} C_VEL
LIN {X 0,Y 270.199,Z 488.415,A -85,B 0,C 180,E1 -17797.036,E2 -17797.036} C_VEL
LIN {X 0,Y 270.29,Z 488.426,A -85,B 0,C 180,E1 -17800.244,E2 -17800.244} C_VEL
LIN {X 0,Y 270.392,Z 488.42,A -85,B 0,C 180,E1 -17804.935,E2 -17804.935} C_VEL
LIN {X 0,Y 270.432,Z 488.415,A -85,B 0,C 180,E1 -17809.519,E2 -17809.519} C_VEL
LIN {X 0,Y 270.601,Z 488.394,A -85,B 0,C 180,E1 -17812.539,E2 -17812.539} C_VEL
LIN {X 0,Y 270.778,Z 488.368,A -85,B 0,C 180,E1 -17818.513,E2 -17818.513} C_VEL
LIN {X 0,Y 270.778,Z 488.38,A -85,B 0,C 180,E1 -17821.487,E2 -17821.487} C_VEL
LIN {X 0,Y 270.6,Z 488.396,A -85,B 0,C 180,E1 -17827.462,E2 -17827.462} C_VEL
LIN {X 0,Y 270.432,Z 488.423,A -85,B 0,C 180,E1 -17830.482,E2 -17830.482} C_VEL
LIN {X 0,Y 270.393,Z 488.429,A -85,B 0,C 180,E1 -17835.065,E2 -17835.065} C_VEL
LIN {X 0,Y 270.292,Z 488.44,A -85,B 0,C 180,E1 -17839.757,E2 -17839.757} C_VEL
LIN {X 0,Y 270.265,Z 488.445,A -85,B 0,C 180,E1 -17844.587,E2 -17844.587} C_VEL
LIN {X 0,Y 270.266,Z 488.443,A -85,B 0,C 180,E1 -17847.91,E2 -17847.91} C_VEL
LIN {X 0,Y 270.177,Z 488.453,A -85,B 0,C 180,E1 -17851.349,E2 -17851.349} C_VEL
LIN {X 0,Y 270.208,Z 488.449,A -85,B 0,C 180,E1 -17854.905,E2 -17854.905} C_VEL
LIN {X 0,Y 270.215,Z 488.454,A -85,B 0,C 180,E1 -17858.719,E2 -17858.719} C_VEL
LIN {X 0,Y 270.196,Z 488.452,A -85,B 0,C 180,E1 -17862.554,E2 -17862.554} C_VEL
LIN {X 0,Y 270.218,Z 488.453,A -85,B 0,C 180,E1 -17867.1,E2 -17867.1} C_VEL
LIN {X 0,Y 270.245,Z 488.587,A -85,B 0,C 180,E1 -17867.459,E2 -17867.459} C_VEL
LIN {X 0,Y 272.544,Z 496.152,A -85,B 0,C 180,E1 -17870.679,E2 -17870.679} C_VEL
LIN {X 0,Y 275.165,Z 506.195,A -85,B 0,C 180,E1 -17874.57,E2 -17874.57} C_VEL
LIN {X 0,Y 277.329,Z 515.328,A -85,B 0,C 180,E1 -17877.85,E2 -17877.85} C_VEL
LIN {X 0,Y 277.816,Z 517.504,A -85,B 0,C 180,E1 -17878.602,E2 -17878.602} C_VEL
LIN {X 0,Y 284.917,Z 533.049,A -85,B 0,C 180,E1 -17879.958,E2 -17879.958} C_VEL
LIN {X 0,Y 289.425,Z 557.14,A -85,B 0,C 180,E1 -17881.153,E2 -17881.153} C_VEL
LIN {X 0,Y 289.715,Z 560.845,A -85,B 0,C 180,E1 -17881.284,E2 -17881.284} C_VEL
LIN {X 0,Y 287.506,Z 633.589,A -85,B 0,C 180,E1 -17882.968,E2 -17882.968} C_VEL
LIN {X 0,Y 286.689,Z 646.612,A -85,B 0,C 180,E1 -17883.524,E2 -17883.524} C_VEL
LIN {X 0,Y 285.394,Z 659.831,A -85,B 0,C 180,E1 -17884.377,E2 -17884.377} C_VEL
LIN {X 0,Y 283.705,Z 672.388,A -85,B 0,C 180,E1 -17885.487,E2 -17885.487} C_VEL
LIN {X 0,Y 281.648,Z 684.19,A -85,B 0,C 180,E1 -17886.86,E2 -17886.86} C_VEL
LIN {X 0,Y 279.753,Z 694.292,A -85,B 0,C 180,E1 -17888.361,E2 -17888.361} C_VEL
LIN {X 0,Y 277.878,Z 703.433,A -85,B 0,C 180,E1 -17890.038,E2 -17890.038} C_VEL
LIN {X 0,Y 275.624,Z 712.914,A -85,B 0,C 180,E1 -17892.185,E2 -17892.185} C_VEL
LIN {X 0,Y 273.761,Z 720.569,A -85,B 0,C 180,E1 -17894.364,E2 -17894.364} C_VEL
LIN {X 0,Y 272.233,Z 726.748,A -85,B 0,C 180,E1 -17896.567,E2 -17896.567} C_VEL
LIN {X 0,Y 270.881,Z 731.717,A -85,B 0,C 180,E1 -17898.781,E2 -17898.781} C_VEL
LIN {X 0,Y 269.932,Z 735.606,A -85,B 0,C 180,E1 -17901.015,E2 -17901.015} C_VEL
LIN {X 0,Y 269.496,Z 737.677,A -85,B 0,C 180,E1 -17902.51,E2 -17902.51} C_VEL
LIN {X 0,Y 269.175,Z 739.315,A -85,B 0,C 180,E1 -17904.007,E2 -17904.007} C_VEL
LIN {X 0,Y 268.659,Z 741.492,A -85,B 0,C 180,E1 -17907.003,E2 -17907.003} C_VEL
LIN {X 0,Y 268.51,Z 742.252,A -85,B 0,C 180,E1 -17910.002,E2 -17910.002} C_VEL
LIN {X 0,Y 268.653,Z 741.549,A -85,B 0,C 180,E1 -17913.001,E2 -17913.001} C_VEL
LIN {X 0,Y 269.157,Z 739.418,A -85,B 0,C 180,E1 -17915.997,E2 -17915.997} C_VEL
LIN {X 0,Y 269.654,Z 737.227,A -85,B 0,C 180,E1 -17917.945,E2 -17917.945} C_VEL
LIN {X 0,Y 270.496,Z 733.313,A -85,B 0,C 180,E1 -17920.481,E2 -17920.481} C_VEL
LIN {X 0,Y 271.712,Z 728.771,A -85,B 0,C 180,E1 -17922.703,E2 -17922.703} C_VEL
LIN {X 0,Y 273.397,Z 721.996,A -85,B 0,C 180,E1 -17925.279,E2 -17925.279} C_VEL
LIN {X 0,Y 275.201,Z 714.709,A -85,B 0,C 180,E1 -17927.464,E2 -17927.464} C_VEL
LIN {X 0,Y 277.451,Z 705.701,A -85,B 0,C 180,E1 -17929.613,E2 -17929.613} C_VEL
LIN {X 0,Y 279.564,Z 695.563,A -85,B 0,C 180,E1 -17931.541,E2 -17931.541} C_VEL
LIN {X 0,Y 281.573,Z 684.955,A -85,B 0,C 180,E1 -17933.15,E2 -17933.15} C_VEL
LIN {X 0,Y 283.614,Z 673.377,A -85,B 0,C 180,E1 -17934.525,E2 -17934.525} C_VEL
LIN {X 0,Y 285.3,Z 661.196,A -85,B 0,C 180,E1 -17935.636,E2 -17935.636} C_VEL
LIN {X 0,Y 286.623,Z 647.701,A -85,B 0,C 180,E1 -17936.535,E2 -17936.535} C_VEL
LIN {X 0,Y 287.59,Z 634.062,A -85,B 0,C 180,E1 -17937.125,E2 -17937.125} C_VEL
LIN {X 0,Y 289.757,Z 558.557,A -85,B 0,C 180,E1 -17938.893,E2 -17938.893} C_VEL
LIN {X 0,Y 284.976,Z 533.281,A -85,B 0,C 180,E1 -17940.15,E2 -17940.15} C_VEL
LIN {X 0,Y 278.662,Z 519.577,A -85,B 0,C 180,E1 -17941.352,E2 -17941.352} C_VEL
LIN {X 0,Y 277.758,Z 517.403,A -85,B 0,C 180,E1 -17941.564,E2 -17941.564} C_VEL
LIN {X 0,Y 275.659,Z 508.118,A -85,B 0,C 180,E1 -17944.853,E2 -17944.853} C_VEL
LIN {X 0,Y 273.447,Z 499.601,A -85,B 0,C 180,E1 -17948.087,E2 -17948.087} C_VEL
LIN {X 0,Y 271.153,Z 491.928,A -85,B 0,C 180,E1 -17951.266,E2 -17951.266} C_VEL
LIN {X 0,Y 270.195,Z 488.456,A -85,B 0,C 180,E1 -17952.813,E2 -17952.813} C_VEL
LIN {X 0,Y 270.178,Z 488.445,A -85,B 0,C 180,E1 -17957.442,E2 -17957.442} C_VEL
LIN {X 0,Y 270.214,Z 488.438,A -85,B 0,C 180,E1 -17961.375,E2 -17961.375} C_VEL
LIN {X 0,Y 270.292,Z 488.534,A -85,B 0,C 180,E1 -17964.937,E2 -17964.937} C_VEL
LIN {X 0,Y 274.455,Z 506.787,A -85,B 0,C 180,E1 -17969.193,E2 -17969.193} C_VEL
LIN {X 0,Y 276.852,Z 518.242,A -85,B 0,C 180,E1 -17971.783,E2 -17971.783} C_VEL
LIN {X 0,Y 276.201,Z 526.931,A -85,B 0,C 180,E1 -17973.564,E2 -17973.564} C_VEL
LIN {X 0,Y 275.717,Z 529.932,A -85,B 0,C 180,E1 -17974.073,E2 -17974.073} C_VEL
LIN {X 0,Y 274.379,Z 534.976,A -85,B 0,C 180,E1 -17974.643,E2 -17974.643} C_VEL
LIN {X 0,Y 272.769,Z 540.381,A -85,B 0,C 180,E1 -17975.037,E2 -17975.037} C_VEL
LIN {X 0,Y 270.983,Z 548.022,A -85,B 0,C 180,E1 -17975.409,E2 -17975.409} C_VEL
LIN {X 0,Y 270.59,Z 553.878,A -85,B 0,C 180,E1 -17975.658,E2 -17975.658} C_VEL
LIN {X 0,Y 270.75,Z 555.821,A -85,B 0,C 180,E1 -17975.748,E2 -17975.748} C_VEL
LIN {X 0,Y 271.521,Z 563.216,A -85,B 0,C 180,E1 -17976.093,E2 -17976.093} C_VEL
LIN {X 0,Y 268.041,Z 648.185,A -85,B 0,C 180,E1 -17979.57,E2 -17979.57} C_VEL
LIN {X 0,Y 267.3,Z 661.41,A -85,B 0,C 180,E1 -17980.413,E2 -17980.413} C_VEL
LIN {X 0,Y 266.492,Z 674.49,A -85,B 0,C 180,E1 -17981.55,E2 -17981.55} C_VEL
LIN {X 0,Y 265.417,Z 687.753,A -85,B 0,C 180,E1 -17983.066,E2 -17983.066} C_VEL
LIN {X 0,Y 264.47,Z 698.41,A -85,B 0,C 180,E1 -17984.589,E2 -17984.589} C_VEL
LIN {X 0,Y 263.683,Z 707.263,A -85,B 0,C 180,E1 -17986.12,E2 -17986.12} C_VEL
LIN {X 0,Y 262.788,Z 718.189,A -85,B 0,C 180,E1 -17988.429,E2 -17988.429} C_VEL
LIN {X 0,Y 262.092,Z 726.896,A -85,B 0,C 180,E1 -17990.741,E2 -17990.741} C_VEL
LIN {X 0,Y 261.627,Z 733.935,A -85,B 0,C 180,E1 -17993.057,E2 -17993.057} C_VEL
LIN {X 0,Y 261.348,Z 739.544,A -85,B 0,C 180,E1 -17995.372,E2 -17995.372} C_VEL
LIN {X 0,Y 261.273,Z 743.854,A -85,B 0,C 180,E1 -17997.687,E2 -17997.687} C_VEL
LIN {X 0,Y 261.222,Z 747.055,A -85,B 0,C 180,E1 -18000,E2 -18000} C_VEL
LIN {X 0,Y 261.349,Z 748.604,A -85,B 0,C 180,E1 -18001.541,E2 -18001.541} C_VEL
LIN {X 0,Y 261.554,Z 749.747,A -85,B 0,C 180,E1 -18003.08,E2 -18003.08} C_VEL
LIN {X 0,Y 261.799,Z 750.463,A -85,B 0,C 180,E1 -18004.619,E2 -18004.619} C_VEL
LIN {X 0,Y 262.12,Z 750.723,A -85,B 0,C 180,E1 -18006.157,E2 -18006.157} C_VEL
LIN {X 0,Y 263.329,Z 750.094,A -85,B 0,C 180,E1 -18009.062,E2 -18009.062} C_VEL
LIN {X 0,Y 264.211,Z 749.039,A -85,B 0,C 180,E1 -18010.731,E2 -18010.731} C_VEL
LIN {X 0,Y 266.263,Z 745.796,A -85,B 0,C 180,E1 -18013.742,E2 -18013.742} C_VEL
LIN {X 0,Y 268.283,Z 742.197,A -85,B 0,C 180,E1 -18015.965,E2 -18015.965} C_VEL
LIN {X 0,Y 270.744,Z 737.458,A -85,B 0,C 180,E1 -18018.149,E2 -18018.149} C_VEL
LIN {X 0,Y 274.001,Z 730.412,A -85,B 0,C 180,E1 -18020.651,E2 -18020.651} C_VEL
LIN {X 0,Y 277.351,Z 722.805,A -85,B 0,C 180,E1 -18022.732,E2 -18022.732} C_VEL
LIN {X 0,Y 281.006,Z 713.441,A -85,B 0,C 180,E1 -18024.766,E2 -18024.766} C_VEL
LIN {X 0,Y 284.32,Z 704.041,A -85,B 0,C 180,E1 -18026.419,E2 -18026.419} C_VEL
LIN {X 0,Y 287.638,Z 693.379,A -85,B 0,C 180,E1 -18027.919,E2 -18027.919} C_VEL
LIN {X 0,Y 290.581,Z 682.758,A -85,B 0,C 180,E1 -18029.127,E2 -18029.127} C_VEL
LIN {X 0,Y 293.421,Z 670.876,A -85,B 0,C 180,E1 -18030.198,E2 -18030.198} C_VEL
LIN {X 0,Y 295.701,Z 659.029,A -85,B 0,C 180,E1 -18031.028,E2 -18031.028} C_VEL
LIN {X 0,Y 297.989,Z 644.703,A -85,B 0,C 180,E1 -18031.751,E2 -18031.751} C_VEL
LIN {X 0,Y 308.149,Z 579.474,A -85,B 0,C 180,E1 -18034.628,E2 -18034.628} C_VEL
LIN {X 0,Y 307.837,Z 568.88,A -85,B 0,C 180,E1 -18036.029,E2 -18036.029} C_VEL
LIN {X 0,Y 306.289,Z 563.797,A -85,B 0,C 180,E1 -18037.571,E2 -18037.571} C_VEL
LIN {X 0,Y 305.017,Z 559.875,A -85,B 0,C 180,E1 -18039.14,E2 -18039.14} C_VEL
LIN {X 0,Y 303.849,Z 556.196,A -85,B 0,C 180,E1 -18041.224,E2 -18041.224} C_VEL
LIN {X 0,Y 303.188,Z 553.887,A -85,B 0,C 180,E1 -18043.732,E2 -18043.732} C_VEL
LIN {X 0,Y 303.264,Z 553.317,A -85,B 0,C 180,E1 -18044.963,E2 -18044.963} C_VEL
LIN {X 0,Y 304.013,Z 553.423,A -85,B 0,C 180,E1 -18047.25,E2 -18047.25} C_VEL
LIN {X 0,Y 305.612,Z 554.797,A -85,B 0,C 180,E1 -18049.492,E2 -18049.492} C_VEL
LIN {X 0,Y 306.565,Z 556.066,A -85,B 0,C 180,E1 -18050.526,E2 -18050.526} C_VEL
LIN {X 0,Y 307.88,Z 563.924,A -85,B 0,C 180,E1 -18052.553,E2 -18052.553} C_VEL
LIN {X 0,Y 307.094,Z 571.998,A -85,B 0,C 180,E1 -18053.24,E2 -18053.24} C_VEL
LIN {X 0,Y 291.047,Z 669.678,A -85,B 0,C 180,E1 -18057.705,E2 -18057.705} C_VEL
LIN {X 0,Y 288.452,Z 683.299,A -85,B 0,C 180,E1 -18058.613,E2 -18058.613} C_VEL
LIN {X 0,Y 285.092,Z 697.319,A -85,B 0,C 180,E1 -18059.847,E2 -18059.847} C_VEL
LIN {X 0,Y 282.107,Z 708.634,A -85,B 0,C 180,E1 -18061.137,E2 -18061.137} C_VEL
LIN {X 0,Y 279.343,Z 718.099,A -85,B 0,C 180,E1 -18062.463,E2 -18062.463} C_VEL
LIN {X 0,Y 275.956,Z 729.086,A -85,B 0,C 180,E1 -18064.343,E2 -18064.343} C_VEL
LIN {X 0,Y 272.494,Z 739.083,A -85,B 0,C 180,E1 -18066.435,E2 -18066.435} C_VEL
LIN {X 0,Y 269.598,Z 747.295,A -85,B 0,C 180,E1 -18068.593,E2 -18068.593} C_VEL
LIN {X 0,Y 266.828,Z 755.181,A -85,B 0,C 180,E1 -18071.175,E2 -18071.175} C_VEL
LIN {X 0,Y 264.687,Z 761.351,A -85,B 0,C 180,E1 -18073.81,E2 -18073.81} C_VEL
LIN {X 0,Y 263.205,Z 765.523,A -85,B 0,C 180,E1 -18076.093,E2 -18076.093} C_VEL
LIN {X 0,Y 261.917,Z 769.534,A -85,B 0,C 180,E1 -18079.172,E2 -18079.172} C_VEL
LIN {X 0,Y 261.512,Z 770.906,A -85,B 0,C 180,E1 -18080.719,E2 -18080.719} C_VEL
LIN {X 0,Y 261.276,Z 771.843,A -85,B 0,C 180,E1 -18082.269,E2 -18082.269} C_VEL
LIN {X 0,Y 261.171,Z 772.503,A -85,B 0,C 180,E1 -18084.656,E2 -18084.656} C_VEL
LIN {X 0,Y 261.281,Z 772.2,A -85,B 0,C 180,E1 -18086.914,E2 -18086.914} C_VEL
LIN {X 0,Y 261.369,Z 772.829,A -85,B 0,C 180,E1 -18089.998,E2 -18089.998} C_VEL
LIN {X 0,Y 261.294,Z 772.064,A -85,B 0,C 180,E1 -18093.082,E2 -18093.082} C_VEL
LIN {X 0,Y 261.248,Z 769.815,A -85,B 0,C 180,E1 -18096.175,E2 -18096.175} C_VEL
LIN {X 0,Y 261.445,Z 766.046,A -85,B 0,C 180,E1 -18099.28,E2 -18099.28} C_VEL
LIN {X 0,Y 262.135,Z 760.665,A -85,B 0,C 180,E1 -18102.383,E2 -18102.383} C_VEL
LIN {X 0,Y 263.233,Z 754.445,A -85,B 0,C 180,E1 -18105.086,E2 -18105.086} C_VEL
LIN {X 0,Y 263.99,Z 750.286,A -85,B 0,C 180,E1 -18106.585,E2 -18106.585} C_VEL
LIN {X 0,Y 265.631,Z 742.684,A -85,B 0,C 180,E1 -18108.909,E2 -18108.909} C_VEL
LIN {X 0,Y 267.576,Z 733.639,A -85,B 0,C 180,E1 -18111.169,E2 -18111.169} C_VEL
LIN {X 0,Y 269.652,Z 724.632,A -85,B 0,C 180,E1 -18113.011,E2 -18113.011} C_VEL
LIN {X 0,Y 272.099,Z 712.774,A -85,B 0,C 180,E1 -18114.994,E2 -18114.994} C_VEL
LIN {X 0,Y 274.405,Z 700.521,A -85,B 0,C 180,E1 -18116.626,E2 -18116.626} C_VEL
LIN {X 0,Y 276.416,Z 688.826,A -85,B 0,C 180,E1 -18117.85,E2 -18117.85} C_VEL
LIN {X 0,Y 278.243,Z 676.096,A -85,B 0,C 180,E1 -18118.884,E2 -18118.884} C_VEL
LIN {X 0,Y 279.803,Z 662.481,A -85,B 0,C 180,E1 -18119.686,E2 -18119.686} C_VEL
LIN {X 0,Y 280.849,Z 648.515,A -85,B 0,C 180,E1 -18120.237,E2 -18120.237} C_VEL
LIN {X 0,Y 283.992,Z 564.159,A -85,B 0,C 180,E1 -18122.454,E2 -18122.454} C_VEL
LIN {X 0,Y 280.825,Z 540.012,A -85,B 0,C 180,E1 -18123.582,E2 -18123.582} C_VEL
LIN {X 0,Y 273.373,Z 523.686,A -85,B 0,C 180,E1 -18125.083,E2 -18125.083} C_VEL
LIN {X 0,Y 272.264,Z 521.034,A -85,B 0,C 180,E1 -18125.356,E2 -18125.356} C_VEL
LIN {X 0,Y 269.731,Z 510.911,A -85,B 0,C 180,E1 -18128.704,E2 -18128.704} C_VEL
LIN {X 0,Y 267.132,Z 501.748,A -85,B 0,C 180,E1 -18131.98,E2 -18131.98} C_VEL
LIN {X 0,Y 264.459,Z 493.372,A -85,B 0,C 180,E1 -18135.233,E2 -18135.233} C_VEL
LIN {X 0,Y 263.193,Z 489.323,A -85,B 0,C 180,E1 -18136.954,E2 -18136.954} C_VEL
LIN {X 0,Y 263.149,Z 489.323,A -85,B 0,C 180,E1 -18140.757,E2 -18140.757} C_VEL
LIN {X 0,Y 263.181,Z 489.293,A -85,B 0,C 180,E1 -18144.021,E2 -18144.021} C_VEL
LIN {X 0,Y 263.125,Z 489.329,A -85,B 0,C 180,E1 -18147.711,E2 -18147.711} C_VEL
LIN {X 0,Y 263.192,Z 489.318,A -85,B 0,C 180,E1 -18151.782,E2 -18151.782} C_VEL
LIN {X 0,Y 263.191,Z 489.318,A -85,B 0,C 180,E1 -18155.211,E2 -18155.211} C_VEL
LIN {X 0,Y 263.252,Z 489.29,A -85,B 0,C 180,E1 -18159.693,E2 -18159.693} C_VEL
LIN {X 0,Y 263.34,Z 489.297,A -85,B 0,C 180,E1 -18164.522,E2 -18164.522} C_VEL
LIN {X 0,Y 263.364,Z 489.293,A -85,B 0,C 180,E1 -18169.234,E2 -18169.234} C_VEL
LIN {X 0,Y 263.562,Z 489.272,A -85,B 0,C 180,E1 -18172.338,E2 -18172.338} C_VEL
LIN {X 0,Y 263.742,Z 489.244,A -85,B 0,C 180,E1 -18178.473,E2 -18178.473} C_VEL
LIN {X 0,Y 263.742,Z 489.256,A -85,B 0,C 180,E1 -18181.527,E2 -18181.527} C_VEL
LIN {X 0,Y 263.562,Z 489.27,A -85,B 0,C 180,E1 -18187.662,E2 -18187.662} C_VEL
LIN {X 0,Y 263.365,Z 489.306,A -85,B 0,C 180,E1 -18190.766,E2 -18190.766} C_VEL
LIN {X 0,Y 263.341,Z 489.307,A -85,B 0,C 180,E1 -18195.479,E2 -18195.479} C_VEL
LIN {X 0,Y 263.254,Z 489.32,A -85,B 0,C 180,E1 -18200.308,E2 -18200.308} C_VEL
LIN {X 0,Y 263.2,Z 489.321,A -85,B 0,C 180,E1 -18205.292,E2 -18205.292} C_VEL
LIN {X 0,Y 263.175,Z 489.327,A -85,B 0,C 180,E1 -18208.73,E2 -18208.73} C_VEL
LIN {X 0,Y 263.126,Z 489.335,A -85,B 0,C 180,E1 -18212.289,E2 -18212.289} C_VEL
LIN {X 0,Y 263.182,Z 489.328,A -85,B 0,C 180,E1 -18215.979,E2 -18215.979} C_VEL
LIN {X 0,Y 263.133,Z 489.33,A -85,B 0,C 180,E1 -18219.868,E2 -18219.868} C_VEL
LIN {X 0,Y 263.137,Z 489.332,A -85,B 0,C 180,E1 -18223.982,E2 -18223.982} C_VEL
LIN {X 0,Y 263.161,Z 489.433,A -85,B 0,C 180,E1 -18226.281,E2 -18226.281} C_VEL
LIN {X 0,Y 265.759,Z 498.023,A -85,B 0,C 180,E1 -18230.077,E2 -18230.077} C_VEL
LIN {X 0,Y 267.962,Z 505.982,A -85,B 0,C 180,E1 -18233.308,E2 -18233.308} C_VEL
LIN {X 0,Y 270.245,Z 515.574,A -85,B 0,C 180,E1 -18236.901,E2 -18236.901} C_VEL
LIN {X 0,Y 270.67,Z 517.579,A -85,B 0,C 180,E1 -18237.614,E2 -18237.614} C_VEL
LIN {X 0,Y 279.159,Z 535.692,A -85,B 0,C 180,E1 -18239.302,E2 -18239.302} C_VEL
LIN {X 0,Y 283.56,Z 559.755,A -85,B 0,C 180,E1 -18240.525,E2 -18240.525} C_VEL
LIN {X 0,Y 281.207,Z 634.672,A -85,B 0,C 180,E1 -18242.312,E2 -18242.312} C_VEL
LIN {X 0,Y 280.399,Z 647.389,A -85,B 0,C 180,E1 -18242.882,E2 -18242.882} C_VEL
LIN {X 0,Y 279.051,Z 660.473,A -85,B 0,C 180,E1 -18243.751,E2 -18243.751} C_VEL
LIN {X 0,Y 277.285,Z 672.948,A -85,B 0,C 180,E1 -18244.881,E2 -18244.881} C_VEL
LIN {X 0,Y 275.158,Z 684.687,A -85,B 0,C 180,E1 -18246.281,E2 -18246.281} C_VEL
LIN {X 0,Y 273.059,Z 695.314,A -85,B 0,C 180,E1 -18247.907,E2 -18247.907} C_VEL
LIN {X 0,Y 271.25,Z 703.882,A -85,B 0,C 180,E1 -18249.528,E2 -18249.528} C_VEL
LIN {X 0,Y 268.903,Z 713.35,A -85,B 0,C 180,E1 -18251.724,E2 -18251.724} C_VEL
LIN {X 0,Y 266.954,Z 720.994,A -85,B 0,C 180,E1 -18253.955,E2 -18253.955} C_VEL
LIN {X 0,Y 265.355,Z 727.166,A -85,B 0,C 180,E1 -18256.212,E2 -18256.212} C_VEL
LIN {X 0,Y 263.924,Z 732.133,A -85,B 0,C 180,E1 -18258.482,E2 -18258.482} C_VEL
LIN {X 0,Y 262.935,Z 736.019,A -85,B 0,C 180,E1 -18260.773,E2 -18260.773} C_VEL
LIN {X 0,Y 262.468,Z 738.088,A -85,B 0,C 180,E1 -18262.308,E2 -18262.308} C_VEL
LIN {X 0,Y 262.143,Z 739.724,A -85,B 0,C 180,E1 -18263.846,E2 -18263.846} C_VEL
LIN {X 0,Y 261.587,Z 741.902,A -85,B 0,C 180,E1 -18266.922,E2 -18266.922} C_VEL
LIN {X 0,Y 261.423,Z 742.661,A -85,B 0,C 180,E1 -18270.002,E2 -18270.002} C_VEL
LIN {X 0,Y 261.581,Z 741.958,A -85,B 0,C 180,E1 -18273.082,E2 -18273.082} C_VEL
LIN {X 0,Y 262.105,Z 739.827,A -85,B 0,C 180,E1 -18276.159,E2 -18276.159} C_VEL
LIN {X 0,Y 262.558,Z 737.92,A -85,B 0,C 180,E1 -18277.946,E2 -18277.946} C_VEL
LIN {X 0,Y 263.52,Z 733.726,A -85,B 0,C 180,E1 -18280.761,E2 -18280.761} C_VEL
LIN {X 0,Y 264.803,Z 729.187,A -85,B 0,C 180,E1 -18283.04,E2 -18283.04} C_VEL
LIN {X 0,Y 266.578,Z 722.415,A -85,B 0,C 180,E1 -18285.68,E2 -18285.68} C_VEL
LIN {X 0,Y 268.46,Z 715.135,A -85,B 0,C 180,E1 -18287.917,E2 -18287.917} C_VEL
LIN {X 0,Y 270.786,Z 706.144,A -85,B 0,C 180,E1 -18290.116,E2 -18290.116} C_VEL
LIN {X 0,Y 272.902,Z 696.462,A -85,B 0,C 180,E1 -18292.012,E2 -18292.012} C_VEL
LIN {X 0,Y 274.825,Z 686.721,A -85,B 0,C 180,E1 -18293.553,E2 -18293.553} C_VEL
LIN {X 0,Y 276.926,Z 675.475,A -85,B 0,C 180,E1 -18294.958,E2 -18294.958} C_VEL
LIN {X 0,Y 278.859,Z 662.877,A -85,B 0,C 180,E1 -18296.172,E2 -18296.172} C_VEL
LIN {X 0,Y 280.157,Z 650.006,A -85,B 0,C 180,E1 -18297.097,E2 -18297.097} C_VEL
LIN {X 0,Y 281.193,Z 637.441,A -85,B 0,C 180,E1 -18297.694,E2 -18297.694} C_VEL
LIN {X 0,Y 281.825,Z 619.955,A -85,B 0,C 180,E1 -18298.182,E2 -18298.182} C_VEL
LIN {X 0,Y 283.614,Z 559.609,A -85,B 0,C 180,E1 -18299.595,E2 -18299.595} C_VEL
LIN {X 0,Y 279.233,Z 535.897,A -85,B 0,C 180,E1 -18300.807,E2 -18300.807} C_VEL
LIN {X 0,Y 272.147,Z 520.827,A -85,B 0,C 180,E1 -18302.208,E2 -18302.208} C_VEL
LIN {X 0,Y 270.639,Z 517.494,A -85,B 0,C 180,E1 -18302.54,E2 -18302.54} C_VEL
LIN {X 0,Y 268.351,Z 507.46,A -85,B 0,C 180,E1 -18306.252,E2 -18306.252} C_VEL
LIN {X 0,Y 265.837,Z 498.327,A -85,B 0,C 180,E1 -18309.943,E2 -18309.943} C_VEL
LIN {X 0,Y 263.113,Z 489.327,A -85,B 0,C 180,E1 -18313.988,E2 -18313.988} C_VEL
LIN {X 0,Y 263.13,Z 489.321,A -85,B 0,C 180,E1 -18318.107,E2 -18318.107} C_VEL
LIN {X 0,Y 263.165,Z 489.313,A -85,B 0,C 180,E1 -18322.104,E2 -18322.104} C_VEL
LIN {X 0,Y 263.218,Z 489.374,A -85,B 0,C 180,E1 -18324.552,E2 -18324.552} C_VEL
LIN {X 0,Y 267.428,Z 507.832,A -85,B 0,C 180,E1 -18328.923,E2 -18328.923} C_VEL
LIN {X 0,Y 269.921,Z 519.584,A -85,B 0,C 180,E1 -18331.629,E2 -18331.629} C_VEL
LIN {X 0,Y 268.626,Z 534.945,A -85,B 0,C 180,E1 -18334.762,E2 -18334.762} C_VEL
LIN {X 0,Y 270.75,Z 555.821,A -85,B 0,C 180,E1 -18335.748,E2 -18335.748} C_VEL
LIN {X 0,Y 270.461,Z 559.669,A -85,B 0,C 180,E1 -18335.897,E2 -18335.897} C_VEL
LIN {X 0,Y 267.898,Z 565.804,A -85,B 0,C 180,E1 -18336.045,E2 -18336.045} C_VEL
LIN {X 0,Y 264.905,Z 571.947,A -85,B 0,C 180,E1 -18336.175,E2 -18336.175} C_VEL
LIN {X 0,Y 264.002,Z 575.855,A -85,B 0,C 180,E1 -18336.307,E2 -18336.307} C_VEL
LIN {X 0,Y 260.985,Z 647.962,A -85,B 0,C 180,E1 -18339.405,E2 -18339.405} C_VEL
LIN {X 0,Y 260.233,Z 661.262,A -85,B 0,C 180,E1 -18340.27,E2 -18340.27} C_VEL
LIN {X 0,Y 259.325,Z 675.466,A -85,B 0,C 180,E1 -18341.544,E2 -18341.544} C_VEL
LIN {X 0,Y 258.243,Z 689.3,A -85,B 0,C 180,E1 -18343.192,E2 -18343.192} C_VEL
LIN {X 0,Y 257.202,Z 700.861,A -85,B 0,C 180,E1 -18344.954,E2 -18344.954} C_VEL
LIN {X 0,Y 256.217,Z 711.36,A -85,B 0,C 180,E1 -18346.921,E2 -18346.921} C_VEL
LIN {X 0,Y 255.499,Z 719.971,A -85,B 0,C 180,E1 -18348.898,E2 -18348.898} C_VEL
LIN {X 0,Y 254.863,Z 728.425,A -85,B 0,C 180,E1 -18351.276,E2 -18351.276} C_VEL
LIN {X 0,Y 254.456,Z 735.198,A -85,B 0,C 180,E1 -18353.657,E2 -18353.657} C_VEL
LIN {X 0,Y 254.261,Z 740.569,A -85,B 0,C 180,E1 -18356.037,E2 -18356.037} C_VEL
LIN {X 0,Y 254.165,Z 744.732,A -85,B 0,C 180,E1 -18358.415,E2 -18358.415} C_VEL
LIN {X 0,Y 254.147,Z 746.907,A -85,B 0,C 180,E1 -18360,E2 -18360} C_VEL
LIN {X 0,Y 254.275,Z 748.628,A -85,B 0,C 180,E1 -18361.584,E2 -18361.584} C_VEL
LIN {X 0,Y 254.488,Z 749.865,A -85,B 0,C 180,E1 -18363.166,E2 -18363.166} C_VEL
LIN {X 0,Y 254.728,Z 750.7,A -85,B 0,C 180,E1 -18364.748,E2 -18364.748} C_VEL
LIN {X 0,Y 255.084,Z 751.141,A -85,B 0,C 180,E1 -18366.327,E2 -18366.327} C_VEL
LIN {X 0,Y 256.293,Z 750.8,A -85,B 0,C 180,E1 -18369.174,E2 -18369.174} C_VEL
LIN {X 0,Y 257.282,Z 749.859,A -85,B 0,C 180,E1 -18371.023,E2 -18371.023} C_VEL
LIN {X 0,Y 258.265,Z 748.634,A -85,B 0,C 180,E1 -18372.574,E2 -18372.574} C_VEL
LIN {X 0,Y 260.188,Z 745.945,A -85,B 0,C 180,E1 -18374.869,E2 -18374.869} C_VEL
LIN {X 0,Y 262.421,Z 742.241,A -85,B 0,C 180,E1 -18377.133,E2 -18377.133} C_VEL
LIN {X 0,Y 265.173,Z 737.439,A -85,B 0,C 180,E1 -18379.347,E2 -18379.347} C_VEL
LIN {X 0,Y 268.737,Z 730.264,A -85,B 0,C 180,E1 -18381.88,E2 -18381.88} C_VEL
LIN {X 0,Y 272.387,Z 722.618,A -85,B 0,C 180,E1 -18383.977,E2 -18383.977} C_VEL
LIN {X 0,Y 276.339,Z 713.159,A -85,B 0,C 180,E1 -18386.021,E2 -18386.021} C_VEL
LIN {X 0,Y 280.292,Z 702.596,A -85,B 0,C 180,E1 -18387.84,E2 -18387.84} C_VEL
LIN {X 0,Y 284.126,Z 690.846,A -85,B 0,C 180,E1 -18389.44,E2 -18389.44} C_VEL
LIN {X 0,Y 287.884,Z 677.483,A -85,B 0,C 180,E1 -18390.841,E2 -18390.841} C_VEL
LIN {X 0,Y 291.069,Z 663.603,A -85,B 0,C 180,E1 -18391.933,E2 -18391.933} C_VEL
LIN {X 0,Y 293.802,Z 648.582,A -85,B 0,C 180,E1 -18392.766,E2 -18392.766} C_VEL
LIN {X 0,Y 304.938,Z 581.926,A -85,B 0,C 180,E1 -18395.748,E2 -18395.748} C_VEL
LIN {X 0,Y 304.905,Z 573.628,A -85,B 0,C 180,E1 -18396.901,E2 -18396.901} C_VEL
LIN {X 0,Y 303.636,Z 568.879,A -85,B 0,C 180,E1 -18398.439,E2 -18398.439} C_VEL
LIN {X 0,Y 302.419,Z 564.84,A -85,B 0,C 180,E1 -18400.296,E2 -18400.296} C_VEL
LIN {X 0,Y 301.752,Z 562.36,A -85,B 0,C 180,E1 -18401.925,E2 -18401.925} C_VEL
LIN {X 0,Y 301.452,Z 560.63,A -85,B 0,C 180,E1 -18404.049,E2 -18404.049} C_VEL
LIN {X 0,Y 301.663,Z 560.144,A -85,B 0,C 180,E1 -18405.657,E2 -18405.657} C_VEL
LIN {X 0,Y 302.462,Z 560.479,A -85,B 0,C 180,E1 -18407.634,E2 -18407.634} C_VEL
LIN {X 0,Y 304.152,Z 562.005,A -85,B 0,C 180,E1 -18409.816,E2 -18409.816} C_VEL
LIN {X 0,Y 304.389,Z 562.884,A -85,B 0,C 180,E1 -18410.187,E2 -18410.187} C_VEL
LIN {X 0,Y 305.01,Z 568.564,A -85,B 0,C 180,E1 -18411.623,E2 -18411.623} C_VEL
LIN {X 0,Y 304.335,Z 573.804,A -85,B 0,C 180,E1 -18412.054,E2 -18412.054} C_VEL
LIN {X 0,Y 287.333,Z 670.103,A -85,B 0,C 180,E1 -18416.503,E2 -18416.503} C_VEL
LIN {X 0,Y 284.514,Z 683.289,A -85,B 0,C 180,E1 -18417.396,E2 -18417.396} C_VEL
LIN {X 0,Y 280.746,Z 697.824,A -85,B 0,C 180,E1 -18418.703,E2 -18418.703} C_VEL
LIN {X 0,Y 277.085,Z 710.031,A -85,B 0,C 180,E1 -18420.149,E2 -18420.149} C_VEL
LIN {X 0,Y 273.81,Z 720.221,A -85,B 0,C 180,E1 -18421.649,E2 -18421.649} C_VEL
LIN {X 0,Y 269.85,Z 731.499,A -85,B 0,C 180,E1 -18423.719,E2 -18423.719} C_VEL
LIN {X 0,Y 266.204,Z 740.934,A -85,B 0,C 180,E1 -18425.843,E2 -18425.843} C_VEL
LIN {X 0,Y 262.657,Z 749.868,A -85,B 0,C 180,E1 -18428.411,E2 -18428.411} C_VEL
LIN {X 0,Y 259.833,Z 757.043,A -85,B 0,C 180,E1 -18431.058,E2 -18431.058} C_VEL
LIN {X 0,Y 257.874,Z 761.99,A -85,B 0,C 180,E1 -18433.37,E2 -18433.37} C_VEL
LIN {X 0,Y 256.322,Z 765.866,A -85,B 0,C 180,E1 -18435.712,E2 -18435.712} C_VEL
LIN {X 0,Y 255.477,Z 767.947,A -85,B 0,C 180,E1 -18437.285,E2 -18437.285} C_VEL
LIN {X 0,Y 254.482,Z 770.787,A -85,B 0,C 180,E1 -18440.46,E2 -18440.46} C_VEL
LIN {X 0,Y 254.214,Z 771.621,A -85,B 0,C 180,E1 -18442.053,E2 -18442.053} C_VEL
LIN {X 0,Y 254.086,Z 772.076,A -85,B 0,C 180,E1 -18444.721,E2 -18444.721} C_VEL
LIN {X 0,Y 254.206,Z 771.667,A -85,B 0,C 180,E1 -18446.828,E2 -18446.828} C_VEL
LIN {X 0,Y 254.225,Z 772.23,A -85,B 0,C 180,E1 -18448.414,E2 -18448.414} C_VEL
LIN {X 0,Y 254.285,Z 772.42,A -85,B 0,C 180,E1 -18449.998,E2 -18449.998} C_VEL
LIN {X 0,Y 254.225,Z 772.222,A -85,B 0,C 180,E1 -18451.582,E2 -18451.582} C_VEL
LIN {X 0,Y 254.198,Z 771.653,A -85,B 0,C 180,E1 -18453.168,E2 -18453.168} C_VEL
LIN {X 0,Y 254.161,Z 769.402,A -85,B 0,C 180,E1 -18456.348,E2 -18456.348} C_VEL
LIN {X 0,Y 254.378,Z 765.629,A -85,B 0,C 180,E1 -18459.54,E2 -18459.54} C_VEL
LIN {X 0,Y 255.163,Z 760.246,A -85,B 0,C 180,E1 -18462.727,E2 -18462.727} C_VEL
LIN {X 0,Y 256.304,Z 754.017,A -85,B 0,C 180,E1 -18465.504,E2 -18465.504} C_VEL
LIN {X 0,Y 257.001,Z 750.443,A -85,B 0,C 180,E1 -18466.84,E2 -18466.84} C_VEL
LIN {X 0,Y 258.867,Z 742.246,A -85,B 0,C 180,E1 -18469.423,E2 -18469.423} C_VEL
LIN {X 0,Y 260.908,Z 733.189,A -85,B 0,C 180,E1 -18471.737,E2 -18471.737} C_VEL
LIN {X 0,Y 263.062,Z 724.164,A -85,B 0,C 180,E1 -18473.622,E2 -18473.622} C_VEL
LIN {X 0,Y 265.517,Z 712.816,A -85,B 0,C 180,E1 -18475.564,E2 -18475.564} C_VEL
LIN {X 0,Y 267.75,Z 701.441,A -85,B 0,C 180,E1 -18477.131,E2 -18477.131} C_VEL
LIN {X 0,Y 270.139,Z 688.246,A -85,B 0,C 180,E1 -18478.555,E2 -18478.555} C_VEL
LIN {X 0,Y 272.037,Z 675.403,A -85,B 0,C 180,E1 -18479.607,E2 -18479.607} C_VEL
LIN {X 0,Y 273.649,Z 661.62,A -85,B 0,C 180,E1 -18480.424,E2 -18480.424} C_VEL
LIN {X 0,Y 274.717,Z 647.275,A -85,B 0,C 180,E1 -18480.985,E2 -18480.985} C_VEL
LIN {X 0,Y 277.894,Z 565.09,A -85,B 0,C 180,E1 -18483.179,E2 -18483.179} C_VEL
LIN {X 0,Y 275.051,Z 542.667,A -85,B 0,C 180,E1 -18484.253,E2 -18484.253} C_VEL
LIN {X 0,Y 266.933,Z 524.86,A -85,B 0,C 180,E1 -18485.962,E2 -18485.962} C_VEL
LIN {X 0,Y 265.11,Z 521.062,A -85,B 0,C 180,E1 -18486.374,E2 -18486.374} C_VEL
LIN {X 0,Y 262.439,Z 510.616,A -85,B 0,C 180,E1 -18489.991,E2 -18489.991} C_VEL
LIN {X 0,Y 259.65,Z 501.079,A -85,B 0,C 180,E1 -18493.611,E2 -18493.611} C_VEL
LIN {X 0,Y 257.091,Z 493.207,A -85,B 0,C 180,E1 -18496.889,E2 -18496.889} C_VEL
LIN {X 0,Y 256.157,Z 490.195,A -85,B 0,C 180,E1 -18498.255,E2 -18498.255} C_VEL
LIN {X 0,Y 256.147,Z 490.176,A -85,B 0,C 180,E1 -18502.87,E2 -18502.87} C_VEL
LIN {X 0,Y 256.076,Z 490.205,A -85,B 0,C 180,E1 -18506.709,E2 -18506.709} C_VEL
LIN {X 0,Y 256.129,Z 490.2,A -85,B 0,C 180,E1 -18511.404,E2 -18511.404} C_VEL
LIN {X 0,Y 256.133,Z 490.185,A -85,B 0,C 180,E1 -18515.696,E2 -18515.696} C_VEL
LIN {X 0,Y 256.152,Z 490.165,A -85,B 0,C 180,E1 -18519.104,E2 -18519.104} C_VEL
LIN {X 0,Y 256.289,Z 490.174,A -85,B 0,C 180,E1 -18524.085,E2 -18524.085} C_VEL
LIN {X 0,Y 256.3,Z 490.172,A -85,B 0,C 180,E1 -18528.934,E2 -18528.934} C_VEL
LIN {X 0,Y 256.53,Z 490.151,A -85,B 0,C 180,E1 -18532.127,E2 -18532.127} C_VEL
LIN {X 0,Y 256.705,Z 490.12,A -85,B 0,C 180,E1 -18538.431,E2 -18538.431} C_VEL
LIN {X 0,Y 256.705,Z 490.133,A -85,B 0,C 180,E1 -18541.569,E2 -18541.569} C_VEL
LIN {X 0,Y 256.53,Z 490.144,A -85,B 0,C 180,E1 -18547.874,E2 -18547.874} C_VEL
LIN {X 0,Y 256.3,Z 490.184,A -85,B 0,C 180,E1 -18551.067,E2 -18551.067} C_VEL
LIN {X 0,Y 256.29,Z 490.186,A -85,B 0,C 180,E1 -18555.916,E2 -18555.916} C_VEL
LIN {X 0,Y 256.157,Z 490.199,A -85,B 0,C 180,E1 -18560.896,E2 -18560.896} C_VEL
LIN {X 0,Y 256.18,Z 490.196,A -85,B 0,C 180,E1 -18565.14,E2 -18565.14} C_VEL
LIN {X 0,Y 256.108,Z 490.201,A -85,B 0,C 180,E1 -18569.601,E2 -18569.601} C_VEL
LIN {X 0,Y 256.078,Z 490.205,A -85,B 0,C 180,E1 -18573.292,E2 -18573.292} C_VEL
LIN {X 0,Y 256.132,Z 490.198,A -85,B 0,C 180,E1 -18577.28,E2 -18577.28} C_VEL
LIN {X 0,Y 256.08,Z 490.211,A -85,B 0,C 180,E1 -18581.199,E2 -18581.199} C_VEL
LIN {X 0,Y 256.07,Z 490.282,A -85,B 0,C 180,E1 -18585.008,E2 -18585.008} C_VEL
LIN {X 0,Y 258.693,Z 498.568,A -85,B 0,C 180,E1 -18588.873,E2 -18588.873} C_VEL
LIN {X 0,Y 260.73,Z 506.013,A -85,B 0,C 180,E1 -18592.039,E2 -18592.039} C_VEL
LIN {X 0,Y 263.163,Z 515.808,A -85,B 0,C 180,E1 -18595.89,E2 -18595.89} C_VEL
LIN {X 0,Y 263.639,Z 517.842,A -85,B 0,C 180,E1 -18596.586,E2 -18596.586} C_VEL
LIN {X 0,Y 272.315,Z 535.978,A -85,B 0,C 180,E1 -18598.395,E2 -18598.395} C_VEL
LIN {X 0,Y 273.591,Z 539.192,A -85,B 0,C 180,E1 -18598.664,E2 -18598.664} C_VEL
LIN {X 0,Y 277.462,Z 560.731,A -85,B 0,C 180,E1 -18599.792,E2 -18599.792} C_VEL
LIN {X 0,Y 275.048,Z 634.552,A -85,B 0,C 180,E1 -18601.584,E2 -18601.584} C_VEL
LIN {X 0,Y 274.189,Z 647.396,A -85,B 0,C 180,E1 -18602.164,E2 -18602.164} C_VEL
LIN {X 0,Y 272.728,Z 661.115,A -85,B 0,C 180,E1 -18603.094,E2 -18603.094} C_VEL
LIN {X 0,Y 270.904,Z 673.499,A -85,B 0,C 180,E1 -18604.246,E2 -18604.246} C_VEL
LIN {X 0,Y 268.69,Z 685.184,A -85,B 0,C 180,E1 -18605.674,E2 -18605.674} C_VEL
LIN {X 0,Y 266.422,Z 696.211,A -85,B 0,C 180,E1 -18607.41,E2 -18607.41} C_VEL
LIN {X 0,Y 264.178,Z 706.081,A -85,B 0,C 180,E1 -18609.362,E2 -18609.362} C_VEL
LIN {X 0,Y 261.824,Z 715.168,A -85,B 0,C 180,E1 -18611.617,E2 -18611.617} C_VEL
LIN {X 0,Y 259.831,Z 722.512,A -85,B 0,C 180,E1 -18613.906,E2 -18613.906} C_VEL
LIN {X 0,Y 257.929,Z 729.341,A -85,B 0,C 180,E1 -18616.611,E2 -18616.611} C_VEL
LIN {X 0,Y 256.569,Z 733.933,A -85,B 0,C 180,E1 -18618.948,E2 -18618.948} C_VEL
LIN {X 0,Y 255.675,Z 737.496,A -85,B 0,C 180,E1 -18621.307,E2 -18621.307} C_VEL
LIN {X 0,Y 255.091,Z 740.135,A -85,B 0,C 180,E1 -18623.675,E2 -18623.675} C_VEL
LIN {X 0,Y 254.518,Z 742.311,A -85,B 0,C 180,E1 -18626.836,E2 -18626.836} C_VEL
LIN {X 0,Y 254.34,Z 743.07,A -85,B 0,C 180,E1 -18630.002,E2 -18630.002} C_VEL
LIN {X 0,Y 254.512,Z 742.366,A -85,B 0,C 180,E1 -18633.168,E2 -18633.168} C_VEL
LIN {X 0,Y 255.058,Z 740.236,A -85,B 0,C 180,E1 -18636.33,E2 -18636.33} C_VEL
LIN {X 0,Y 255.489,Z 738.536,A -85,B 0,C 180,E1 -18637.988,E2 -18637.988} C_VEL
LIN {X 0,Y 256.224,Z 735.417,A -85,B 0,C 180,E1 -18640.272,E2 -18640.272} C_VEL
LIN {X 0,Y 257.415,Z 731.225,A -85,B 0,C 180,E1 -18642.618,E2 -18642.618} C_VEL
LIN {X 0,Y 259.2,Z 724.961,A -85,B 0,C 180,E1 -18645.331,E2 -18645.331} C_VEL
LIN {X 0,Y 261.084,Z 718.183,A -85,B 0,C 180,E1 -18647.63,E2 -18647.63} C_VEL
LIN {X 0,Y 262.909,Z 711.313,A -85,B 0,C 180,E1 -18649.523,E2 -18649.523} C_VEL
LIN {X 0,Y 265,Z 703.099,A -85,B 0,C 180,E1 -18651.389,E2 -18651.389} C_VEL
LIN {X 0,Y 267.153,Z 693.13,A -85,B 0,C 180,E1 -18653.243,E2 -18653.243} C_VEL
LIN {X 0,Y 269.432,Z 681.923,A -85,B 0,C 180,E1 -18654.875,E2 -18654.875} C_VEL
LIN {X 0,Y 271.399,Z 671.026,A -85,B 0,C 180,E1 -18656.12,E2 -18656.12} C_VEL
LIN {X 0,Y 273.07,Z 659.051,A -85,B 0,C 180,E1 -18657.185,E2 -18657.185} C_VEL
LIN {X 0,Y 274.342,Z 646.127,A -85,B 0,C 180,E1 -18658.031,E2 -18658.031} C_VEL
LIN {X 0,Y 275.261,Z 633.675,A -85,B 0,C 180,E1 -18658.552,E2 -18658.552} C_VEL
LIN {X 0,Y 277.557,Z 560.693,A -85,B 0,C 180,E1 -18660.323,E2 -18660.323} C_VEL
LIN {X 0,Y 273.513,Z 538.758,A -85,B 0,C 180,E1 -18661.485,E2 -18661.485} C_VEL
LIN {X 0,Y 266.913,Z 524.631,A -85,B 0,C 180,E1 -18662.845,E2 -18662.845} C_VEL
LIN {X 0,Y 263.533,Z 517.548,A -85,B 0,C 180,E1 -18663.602,E2 -18663.602} C_VEL
LIN {X 0,Y 261.184,Z 507.581,A -85,B 0,C 180,E1 -18667.459,E2 -18667.459} C_VEL
LIN {X 0,Y 258.725,Z 498.952,A -85,B 0,C 180,E1 -18671.117,E2 -18671.117} C_VEL
LIN {X 0,Y 257.066,Z 493.6,A -85,B 0,C 180,E1 -18673.574,E2 -18673.574} C_VEL
LIN {X 0,Y 256.039,Z 490.211,A -85,B 0,C 180,E1 -18675.213,E2 -18675.213} C_VEL
LIN {X 0,Y 256.061,Z 490.205,A -85,B 0,C 180,E1 -18678.797,E2 -18678.797} C_VEL
LIN {X 0,Y 256.137,Z 490.191,A -85,B 0,C 180,E1 -18682.868,E2 -18682.868} C_VEL
LIN {X 0,Y 256.188,Z 490.308,A -85,B 0,C 180,E1 -18684.182,E2 -18684.182} C_VEL
LIN {X 0,Y 260.204,Z 507.962,A -85,B 0,C 180,E1 -18688.445,E2 -18688.445} C_VEL
LIN {X 0,Y 262.829,Z 519.87,A -85,B 0,C 180,E1 -18691.228,E2 -18691.228} C_VEL
LIN {X 0,Y 262.375,Z 527.768,A -85,B 0,C 180,E1 -18692.911,E2 -18692.911} C_VEL
LIN {X 0,Y 261.698,Z 534.975,A -85,B 0,C 180,E1 -18694.419,E2 -18694.419} C_VEL
LIN {X 0,Y 263.816,Z 556.71,A -85,B 0,C 180,E1 -18695.469,E2 -18695.469} C_VEL
LIN {X 0,Y 264.561,Z 563.938,A -85,B 0,C 180,E1 -18695.816,E2 -18695.816} C_VEL
LIN {X 0,Y 264.002,Z 575.855,A -85,B 0,C 180,E1 -18696.307,E2 -18696.307} C_VEL
LIN {X 0,Y 262.971,Z 581.596,A -85,B 0,C 180,E1 -18696.517,E2 -18696.517} C_VEL
LIN {X 0,Y 256.519,Z 600.128,A -85,B 0,C 180,E1 -18697.12,E2 -18697.12} C_VEL
LIN {X 0,Y 255.657,Z 605.87,A -85,B 0,C 180,E1 -18697.353,E2 -18697.353} C_VEL
LIN {X 0,Y 253.857,Z 649.461,A -85,B 0,C 180,E1 -18699.33,E2 -18699.33} C_VEL
LIN {X 0,Y 253.061,Z 663.604,A -85,B 0,C 180,E1 -18700.322,E2 -18700.322} C_VEL
LIN {X 0,Y 252.105,Z 677.162,A -85,B 0,C 180,E1 -18701.62,E2 -18701.62} C_VEL
LIN {X 0,Y 251.143,Z 689.333,A -85,B 0,C 180,E1 -18703.122,E2 -18703.122} C_VEL
LIN {X 0,Y 250.115,Z 700.939,A -85,B 0,C 180,E1 -18704.935,E2 -18704.935} C_VEL
LIN {X 0,Y 249.115,Z 711.425,A -85,B 0,C 180,E1 -18706.956,E2 -18706.956} C_VEL
LIN {X 0,Y 248.303,Z 721.59,A -85,B 0,C 180,E1 -18709.398,E2 -18709.398} C_VEL
LIN {X 0,Y 247.681,Z 729.792,A -85,B 0,C 180,E1 -18711.843,E2 -18711.843} C_VEL
LIN {X 0,Y 247.247,Z 736.974,A -85,B 0,C 180,E1 -18714.55,E2 -18714.55} C_VEL
LIN {X 0,Y 247.138,Z 741.591,A -85,B 0,C 180,E1 -18716.739,E2 -18716.739} C_VEL
LIN {X 0,Y 247.059,Z 745.6,A -85,B 0,C 180,E1 -18719.185,E2 -18719.185} C_VEL
LIN {X 0,Y 247.203,Z 748.527,A -85,B 0,C 180,E1 -18721.629,E2 -18721.629} C_VEL
LIN {X 0,Y 247.424,Z 749.952,A -85,B 0,C 180,E1 -18723.256,E2 -18723.256} C_VEL
LIN {X 0,Y 247.662,Z 750.912,A -85,B 0,C 180,E1 -18724.883,E2 -18724.883} C_VEL
LIN {X 0,Y 248.032,Z 751.468,A -85,B 0,C 180,E1 -18726.508,E2 -18726.508} C_VEL
LIN {X 0,Y 249.256,Z 751.453,A -85,B 0,C 180,E1 -18729.29,E2 -18729.29} C_VEL
LIN {X 0,Y 250.371,Z 750.658,A -85,B 0,C 180,E1 -18731.332,E2 -18731.332} C_VEL
LIN {X 0,Y 252.671,Z 748.067,A -85,B 0,C 180,E1 -18734.497,E2 -18734.497} C_VEL
LIN {X 0,Y 254.953,Z 744.998,A -85,B 0,C 180,E1 -18736.824,E2 -18736.824} C_VEL
LIN {X 0,Y 257.691,Z 740.859,A -85,B 0,C 180,E1 -18739.103,E2 -18739.103} C_VEL
LIN {X 0,Y 261.322,Z 734.612,A -85,B 0,C 180,E1 -18741.703,E2 -18741.703} C_VEL
LIN {X 0,Y 264.963,Z 727.854,A -85,B 0,C 180,E1 -18743.859,E2 -18743.859} C_VEL
LIN {X 0,Y 269.01,Z 719.581,A -85,B 0,C 180,E1 -18745.951,E2 -18745.951} C_VEL
LIN {X 0,Y 273.396,Z 709.432,A -85,B 0,C 180,E1 -18747.978,E2 -18747.978} C_VEL
LIN {X 0,Y 277.731,Z 698.038,A -85,B 0,C 180,E1 -18749.776,E2 -18749.776} C_VEL
LIN {X 0,Y 281.555,Z 686.55,A -85,B 0,C 180,E1 -18751.195,E2 -18751.195} C_VEL
LIN {X 0,Y 285.216,Z 673.769,A -85,B 0,C 180,E1 -18752.408,E2 -18752.408} C_VEL
LIN {X 0,Y 287.995,Z 661.812,A -85,B 0,C 180,E1 -18753.303,E2 -18753.303} C_VEL
LIN {X 0,Y 290.767,Z 646.888,A -85,B 0,C 180,E1 -18754.087,E2 -18754.087} C_VEL
LIN {X 0,Y 302.003,Z 584.363,A -85,B 0,C 180,E1 -18756.913,E2 -18756.913} C_VEL
LIN {X 0,Y 302.129,Z 578.673,A -85,B 0,C 180,E1 -18757.729,E2 -18757.729} C_VEL
LIN {X 0,Y 301.178,Z 574.463,A -85,B 0,C 180,E1 -18759.179,E2 -18759.179} C_VEL
LIN {X 0,Y 300.179,Z 570.308,A -85,B 0,C 180,E1 -18761.267,E2 -18761.267} C_VEL
LIN {X 0,Y 299.703,Z 568.219,A -85,B 0,C 180,E1 -18763.097,E2 -18763.097} C_VEL
LIN {X 0,Y 299.819,Z 567.037,A -85,B 0,C 180,E1 -18765.312,E2 -18765.312} C_VEL
LIN {X 0,Y 300.662,Z 567.316,A -85,B 0,C 180,E1 -18767.564,E2 -18767.564} C_VEL
LIN {X 0,Y 302.083,Z 568.689,A -85,B 0,C 180,E1 -18769.54,E2 -18769.54} C_VEL
LIN {X 0,Y 302.361,Z 572.676,A -85,B 0,C 180,E1 -18770.601,E2 -18770.601} C_VEL
LIN {X 0,Y 301.814,Z 576.103,A -85,B 0,C 180,E1 -18770.854,E2 -18770.854} C_VEL
LIN {X 0,Y 284.081,Z 669.802,A -85,B 0,C 180,E1 -18775.209,E2 -18775.209} C_VEL
LIN {X 0,Y 281.041,Z 682.733,A -85,B 0,C 180,E1 -18776.083,E2 -18776.083} C_VEL
LIN {X 0,Y 277.047,Z 696.961,A -85,B 0,C 180,E1 -18777.355,E2 -18777.355} C_VEL
LIN {X 0,Y 273.043,Z 709.2,A -85,B 0,C 180,E1 -18778.799,E2 -18778.799} C_VEL
LIN {X 0,Y 269.068,Z 720.419,A -85,B 0,C 180,E1 -18780.459,E2 -18780.459} C_VEL
LIN {X 0,Y 264.467,Z 732.304,A -85,B 0,C 180,E1 -18782.714,E2 -18782.714} C_VEL
LIN {X 0,Y 260.546,Z 741.395,A -85,B 0,C 180,E1 -18784.857,E2 -18784.857} C_VEL
LIN {X 0,Y 256.691,Z 750.098,A -85,B 0,C 180,E1 -18787.459,E2 -18787.459} C_VEL
LIN {X 0,Y 253.986,Z 756.178,A -85,B 0,C 180,E1 -18789.762,E2 -18789.762} C_VEL
LIN {X 0,Y 251.718,Z 761.147,A -85,B 0,C 180,E1 -18792.112,E2 -18792.112} C_VEL
LIN {X 0,Y 249.979,Z 765.092,A -85,B 0,C 180,E1 -18794.507,E2 -18794.507} C_VEL
LIN {X 0,Y 248.518,Z 768.088,A -85,B 0,C 180,E1 -18796.922,E2 -18796.922} C_VEL
LIN {X 0,Y 247.437,Z 770.684,A -85,B 0,C 180,E1 -18800.186,E2 -18800.186} C_VEL
LIN {X 0,Y 247.153,Z 771.351,A -85,B 0,C 180,E1 -18801.824,E2 -18801.824} C_VEL
LIN {X 0,Y 247.059,Z 771.481,A -85,B 0,C 180,E1 -18805.102,E2 -18805.102} C_VEL
LIN {X 0,Y 247.134,Z 771.258,A -85,B 0,C 180,E1 -18806.737,E2 -18806.737} C_VEL
LIN {X 0,Y 247.148,Z 771.821,A -85,B 0,C 180,E1 -18808.368,E2 -18808.368} C_VEL
LIN {X 0,Y 247.205,Z 772.012,A -85,B 0,C 180,E1 -18809.998,E2 -18809.998} C_VEL
LIN {X 0,Y 247.148,Z 771.813,A -85,B 0,C 180,E1 -18811.627,E2 -18811.627} C_VEL
LIN {X 0,Y 247.106,Z 771.243,A -85,B 0,C 180,E1 -18813.259,E2 -18813.259} C_VEL
